Yaskawa INFORM job: vendrediTRJ1.JBI

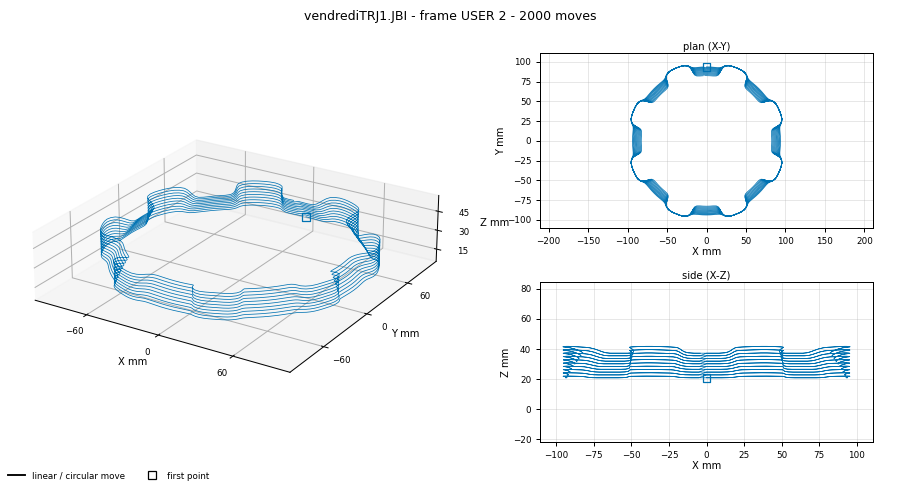
[picture p0: tool path of vendrediTRJ1.JBI in frame USER 2, 2000 of 2000 moves have a stored position in this frame; points joined in program order, loops and branches not executed]
/JOB
//NAME temp/vendrediTRJ1
///FOLDERNAME DEMO
//POS
///NPOS 2000,0,2000,0,0,0
///USER 2
///TOOL 7
///POSTYPE USER
///RECTAN
///RCONF 1,0,0,0,0,0,0,0,0,0,0,0,0,0,0,0,0,0,0,0,0,0,0,0
C00000=0.000,93.772,20.859,-180.0000,28.8281,-3690.0000
C00001=5.223,93.624,20.857,-179.9587,28.8401,-3693.1930
C00002=10.031,93.243,20.860,179.4696,28.7637,-3696.1402
C00003=14.399,92.874,20.935,176.5083,27.4530,-3698.8129
C00004=17.292,92.935,21.118,171.4736,22.1760,-3700.5402
C00005=19.271,93.399,21.361,170.6019,14.0567,-3701.6582
C00006=20.902,94.108,21.598,173.3176,8.0331,-3702.5225
C00007=22.556,94.852,21.773,176.3408,5.3244,-3703.3766
C00008=24.607,95.353,21.858,178.5800,3.6143,-3704.4702
C00009=27.423,95.407,21.902,179.6582,1.5415,-3706.0363
C00010=30.651,94.973,21.938,179.9852,0.1578,-3707.8866
C00011=33.828,94.073,21.973,-179.9998,0.0671,-3709.7782
C00012=36.813,92.974,21.997,179.9979,0.0053,-3711.6011
C00013=39.712,91.773,21.997,-179.9970,0.0075,-3713.3991
C00014=42.599,90.440,21.973,179.9991,0.0692,-3715.2213
C00015=45.483,88.829,21.938,-179.9836,0.1565,-3717.1138
C00016=48.072,86.854,21.902,-179.6591,1.5379,-3718.9637
C00017=50.025,84.825,21.858,-178.5802,3.6128,-3720.5297
C00018=51.121,83.020,21.773,-176.3413,5.3283,-3721.6234
C00019=51.765,81.324,21.598,-173.3148,8.0333,-3722.4779
C00020=52.416,79.670,21.361,-170.5989,14.0579,-3723.3415
C00021=53.488,77.942,21.118,-171.4764,22.1779,-3724.4600
C00022=55.491,75.854,20.935,-176.5044,27.4539,-3726.1873
C00023=58.840,73.026,20.860,-179.4708,28.7627,-3728.8598
C00024=62.509,69.895,20.857,179.9582,28.8407,-3731.8071
C00025=66.307,66.307,20.859,180.0000,28.8305,-3735.0000
C00026=69.895,62.509,20.857,-179.9582,28.8407,-3738.1929
C00027=73.026,58.840,20.860,179.4708,28.7627,-3741.1402
C00028=75.854,55.491,20.935,176.5044,27.4539,-3743.8127
C00029=77.942,53.488,21.118,171.4764,22.1779,-3745.5400
C00030=79.670,52.416,21.361,170.5989,14.0579,-3746.6585
C00031=81.324,51.765,21.598,173.3148,8.0333,-3747.5221
C00032=83.020,51.121,21.773,176.3413,5.3283,-3748.3766
C00033=84.825,50.025,21.858,178.5802,3.6128,-3749.4703
C00034=86.854,48.072,21.902,179.6591,1.5379,-3751.0363
C00035=88.829,45.483,21.938,179.9836,0.1565,-3752.8862
C00036=90.440,42.599,21.973,-179.9991,0.0692,-3754.7787
C00037=91.773,39.712,21.997,179.9970,0.0075,-3756.6009
C00038=92.974,36.813,21.997,-179.9979,0.0053,-3758.3989
C00039=94.073,33.828,21.973,179.9998,0.0671,-3760.2218
C00040=94.973,30.651,21.938,-179.9852,0.1578,-3762.1134
C00041=95.407,27.423,21.902,-179.6582,1.5415,-3763.9637
C00042=95.353,24.607,21.858,-178.5800,3.6143,-3765.5298
C00043=94.852,22.556,21.773,-176.3408,5.3244,-3766.6234
C00044=94.108,20.902,21.598,-173.3176,8.0331,-3767.4775
C00045=93.399,19.271,21.361,-170.6019,14.0567,-3768.3418
C00046=92.935,17.292,21.118,-171.4736,22.1760,-3769.4598
C00047=92.874,14.399,20.935,-176.5083,27.4530,-3771.1871
C00048=93.243,10.031,20.860,-179.4696,28.7637,-3773.8598
C00049=93.624,5.223,20.857,179.9587,28.8401,-3776.8070
C00050=93.772,0.000,20.859,180.0000,28.8281,-3780.0000
C00051=93.624,-5.223,20.857,-179.9587,28.8401,-3783.1930
C00052=93.243,-10.031,20.860,179.4696,28.7637,-3786.1402
C00053=92.875,-14.399,20.935,176.5083,27.4530,-3788.8128
C00054=92.935,-17.292,21.118,171.4736,22.1760,-3790.5402
C00055=93.399,-19.271,21.361,170.6019,14.0567,-3791.6582
C00056=94.108,-20.902,21.598,173.3176,8.0331,-3792.5225
C00057=94.852,-22.556,21.773,176.3408,5.3244,-3793.3766
C00058=95.353,-24.607,21.858,178.5800,3.6143,-3794.4702
C00059=95.407,-27.423,21.902,179.6582,1.5415,-3796.0363
C00060=94.973,-30.651,21.938,179.9852,0.1578,-3797.8866
C00061=94.073,-33.828,21.973,-179.9998,0.0671,-3799.7782
C00062=92.974,-36.813,21.997,179.9979,0.0053,-3801.6011
C00063=91.773,-39.712,21.997,-179.9970,0.0075,-3803.3991
C00064=90.440,-42.599,21.973,179.9991,0.0692,-3805.2213
C00065=88.829,-45.483,21.938,-179.9836,0.1565,-3807.1138
C00066=86.854,-48.072,21.902,-179.6591,1.5379,-3808.9637
C00067=84.825,-50.025,21.858,-178.5802,3.6128,-3810.5297
C00068=83.020,-51.121,21.773,-176.3413,5.3283,-3811.6234
C00069=81.324,-51.765,21.598,-173.3148,8.0333,-3812.4779
C00070=79.670,-52.416,21.361,-170.5989,14.0579,-3813.3415
C00071=77.942,-53.488,21.118,-171.4764,22.1779,-3814.4600
C00072=75.854,-55.491,20.935,-176.5044,27.4539,-3816.1873
C00073=73.026,-58.840,20.860,-179.4708,28.7627,-3818.8598
C00074=69.895,-62.509,20.857,179.9582,28.8407,-3821.8071
C00075=66.307,-66.307,20.859,-180.0000,28.8305,-3825.0000
C00076=62.509,-69.895,20.857,-179.9582,28.8407,-3828.1929
C00077=58.840,-73.026,20.860,179.4708,28.7627,-3831.1402
C00078=55.491,-75.854,20.935,176.5044,27.4539,-3833.8127
C00079=53.488,-77.942,21.118,171.4764,22.1779,-3835.5400
C00080=52.416,-79.670,21.361,170.5989,14.0579,-3836.6585
C00081=51.765,-81.324,21.598,173.3148,8.0333,-3837.5221
C00082=51.121,-83.020,21.773,176.3413,5.3283,-3838.3766
C00083=50.025,-84.825,21.858,178.5802,3.6128,-3839.4703
C00084=48.072,-86.854,21.902,179.6591,1.5379,-3841.0363
C00085=45.483,-88.829,21.938,179.9836,0.1565,-3842.8862
C00086=42.599,-90.440,21.973,-179.9991,0.0692,-3844.7787
C00087=39.712,-91.773,21.997,179.9970,0.0075,-3846.6009
C00088=36.813,-92.974,21.997,-179.9979,0.0053,-3848.3989
C00089=33.828,-94.073,21.973,179.9998,0.0671,-3850.2218
C00090=30.651,-94.973,21.938,-179.9852,0.1578,-3852.1134
C00091=27.423,-95.407,21.902,-179.6582,1.5415,-3853.9637
C00092=24.607,-95.353,21.858,-178.5800,3.6143,-3855.5298
C00093=22.556,-94.852,21.773,-176.3408,5.3244,-3856.6234
C00094=20.902,-94.108,21.598,-173.3176,8.0331,-3857.4775
C00095=19.271,-93.399,21.361,-170.6019,14.0567,-3858.3418
C00096=17.292,-92.935,21.118,-171.4736,22.1760,-3859.4598
C00097=14.399,-92.874,20.935,-176.5083,27.4530,-3861.1871
C00098=10.031,-93.243,20.860,-179.4696,28.7637,-3863.8598
C00099=5.223,-93.624,20.857,179.9587,28.8401,-3866.8070
C00100=0.000,-93.772,20.859,-180.0000,28.8281,-3870.0000
C00101=-5.223,-93.624,20.857,-179.9587,28.8401,-3873.1930
C00102=-10.031,-93.243,20.860,179.4696,28.7637,-3876.1402
C00103=-14.399,-92.875,20.935,176.5083,27.4530,-3878.8128
C00104=-17.292,-92.935,21.118,171.4736,22.1760,-3880.5402
C00105=-19.271,-93.399,21.361,170.6019,14.0567,-3881.6582
C00106=-20.902,-94.108,21.598,173.3176,8.0331,-3882.5225
C00107=-22.556,-94.852,21.773,176.3408,5.3244,-3883.3766
C00108=-24.607,-95.353,21.858,178.5800,3.6143,-3884.4702
C00109=-27.423,-95.407,21.902,179.6582,1.5415,-3886.0363
C00110=-30.651,-94.973,21.938,179.9852,0.1578,-3887.8866
C00111=-33.828,-94.073,21.973,-179.9998,0.0671,-3889.7782
C00112=-36.813,-92.974,21.997,179.9979,0.0053,-3891.6011
C00113=-39.712,-91.773,21.997,-179.9970,0.0075,-3893.3991
C00114=-42.599,-90.440,21.973,179.9991,0.0692,-3895.2213
C00115=-45.483,-88.829,21.938,-179.9836,0.1565,-3897.1138
C00116=-48.072,-86.854,21.902,-179.6591,1.5379,-3898.9637
C00117=-50.025,-84.825,21.858,-178.5802,3.6128,-3900.5297
C00118=-51.121,-83.020,21.773,-176.3413,5.3283,-3901.6234
C00119=-51.765,-81.324,21.598,-173.3148,8.0333,-3902.4779
C00120=-52.416,-79.670,21.361,-170.5989,14.0579,-3903.3415
C00121=-53.488,-77.942,21.118,-171.4764,22.1779,-3904.4600
C00122=-55.491,-75.854,20.935,-176.5044,27.4539,-3906.1873
C00123=-58.840,-73.026,20.860,-179.4708,28.7627,-3908.8598
C00124=-62.509,-69.895,20.857,179.9582,28.8407,-3911.8071
C00125=-66.307,-66.307,20.859,-180.0000,28.8305,-3915.0000
C00126=-69.895,-62.509,20.857,-179.9582,28.8407,-3918.1929
C00127=-73.026,-58.840,20.860,179.4708,28.7627,-3921.1402
C00128=-75.854,-55.491,20.935,176.5044,27.4539,-3923.8127
C00129=-77.942,-53.488,21.118,171.4764,22.1779,-3925.5400
C00130=-79.670,-52.416,21.361,170.5989,14.0579,-3926.6585
C00131=-81.324,-51.765,21.598,173.3148,8.0333,-3927.5221
C00132=-83.020,-51.121,21.773,176.3413,5.3283,-3928.3766
C00133=-84.825,-50.025,21.858,178.5802,3.6128,-3929.4703
C00134=-86.854,-48.072,21.902,179.6591,1.5379,-3931.0363
C00135=-88.829,-45.483,21.938,179.9836,0.1565,-3932.8862
C00136=-90.440,-42.599,21.973,-179.9991,0.0692,-3934.7787
C00137=-91.773,-39.712,21.997,179.9970,0.0075,-3936.6009
C00138=-92.974,-36.813,21.997,-179.9979,0.0053,-3938.3989
C00139=-94.073,-33.828,21.973,179.9998,0.0671,-3940.2218
C00140=-94.973,-30.651,21.938,-179.9852,0.1578,-3942.1134
C00141=-95.407,-27.423,21.902,-179.6582,1.5415,-3943.9637
C00142=-95.353,-24.607,21.858,-178.5800,3.6143,-3945.5298
C00143=-94.852,-22.556,21.773,-176.3408,5.3244,-3946.6234
C00144=-94.108,-20.902,21.598,-173.3176,8.0331,-3947.4775
C00145=-93.399,-19.271,21.361,-170.6019,14.0567,-3948.3418
C00146=-92.935,-17.292,21.118,-171.4736,22.1760,-3949.4598
C00147=-92.874,-14.399,20.935,-176.5083,27.4530,-3951.1871
C00148=-93.243,-10.031,20.860,-179.4696,28.7637,-3953.8598
C00149=-93.624,-5.223,20.857,179.9587,28.8401,-3956.8070
C00150=-93.772,0.000,20.859,180.0000,28.8281,-3960.0000
C00151=-93.624,5.223,20.857,-179.9587,28.8401,-3963.1930
C00152=-93.243,10.031,20.860,179.4696,28.7637,-3966.1402
C00153=-92.875,14.399,20.935,176.5083,27.4530,-3968.8128
C00154=-92.935,17.292,21.118,171.4736,22.1760,-3970.5402
C00155=-93.399,19.271,21.361,170.6019,14.0567,-3971.6582
C00156=-94.108,20.902,21.598,173.3176,8.0331,-3972.5225
C00157=-94.852,22.556,21.773,176.3408,5.3244,-3973.3766
C00158=-95.353,24.607,21.858,178.5800,3.6143,-3974.4702
C00159=-95.407,27.423,21.902,179.6582,1.5415,-3976.0363
C00160=-94.973,30.651,21.938,179.9852,0.1578,-3977.8866
C00161=-94.073,33.828,21.973,-179.9998,0.0671,-3979.7782
C00162=-92.974,36.813,21.997,179.9979,0.0053,-3981.6011
C00163=-91.773,39.712,21.997,-179.9970,0.0075,-3983.3991
C00164=-90.440,42.599,21.973,179.9991,0.0692,-3985.2213
C00165=-88.829,45.483,21.938,-179.9836,0.1565,-3987.1138
C00166=-86.854,48.072,21.902,-179.6591,1.5379,-3988.9637
C00167=-84.825,50.025,21.858,-178.5802,3.6128,-3990.5297
C00168=-83.020,51.121,21.773,-176.3413,5.3283,-3991.6234
C00169=-81.324,51.765,21.598,-173.3148,8.0333,-3992.4779
C00170=-79.670,52.416,21.361,-170.5989,14.0579,-3993.3415
C00171=-77.942,53.488,21.118,-171.4764,22.1779,-3994.4600
C00172=-75.854,55.491,20.935,-176.5044,27.4539,-3996.1873
C00173=-73.026,58.840,20.860,-179.4708,28.7627,-3998.8598
C00174=-69.895,62.509,20.857,179.9582,28.8407,-4001.8071
C00175=-66.307,66.307,20.859,180.0000,28.8305,-4005.0000
C00176=-62.509,69.895,20.857,-179.9582,28.8407,-4008.1929
C00177=-58.840,73.026,20.860,179.4708,28.7627,-4011.1402
C00178=-55.491,75.854,20.935,176.5044,27.4539,-4013.8127
C00179=-53.488,77.942,21.118,171.4764,22.1779,-4015.5400
C00180=-52.416,79.670,21.361,170.5989,14.0579,-4016.6585
C00181=-51.765,81.324,21.598,173.3148,8.0333,-4017.5221
C00182=-51.121,83.020,21.773,176.3413,5.3283,-4018.3766
C00183=-50.025,84.825,21.858,178.5802,3.6128,-4019.4703
C00184=-48.072,86.854,21.902,179.6591,1.5379,-4021.0363
C00185=-45.483,88.829,21.938,179.9836,0.1565,-4022.8862
C00186=-42.599,90.440,21.973,-179.9991,0.0692,-4024.7787
C00187=-39.712,91.773,21.997,179.9970,0.0075,-4026.6009
C00188=-36.813,92.974,21.997,-179.9979,0.0053,-4028.3989
C00189=-33.828,94.073,21.973,179.9998,0.0671,-4030.2218
C00190=-30.651,94.973,21.938,-179.9852,0.1578,-4032.1134
C00191=-27.423,95.407,21.902,-179.6582,1.5415,-4033.9637
C00192=-24.607,95.353,21.858,-178.5800,3.6143,-4035.5298
C00193=-22.556,94.852,21.773,-176.3408,5.3244,-4036.6234
C00194=-20.902,94.108,21.598,-173.3176,8.0331,-4037.4775
C00195=-19.271,93.399,21.361,-170.6019,14.0567,-4038.3418
C00196=-17.292,92.935,21.118,-171.4736,22.1760,-4039.4598
C00197=-14.399,92.875,20.935,-176.5083,27.4530,-4041.1872
C00198=-10.031,93.243,20.860,-179.4696,28.7637,-4043.8598
C00199=-5.223,93.624,20.857,179.9587,28.8401,-4046.8070
C00200=0.000,92.684,22.771,-180.0000,30.3909,-4050.0000
C00201=5.124,92.540,22.769,-179.9518,30.3994,-4053.1693
C00202=9.864,92.169,22.773,179.3255,30.3134,-4056.1086
C00203=14.194,91.838,22.865,175.6033,28.8062,-4058.7858
C00204=17.042,91.994,23.091,169.6619,22.2216,-4060.4951
C00205=18.986,92.606,23.393,169.6266,12.7358,-4061.5862
C00206=20.592,93.503,23.691,173.2393,6.5920,-4062.4199
C00207=22.223,94.456,23.912,176.4053,4.2313,-4063.2394
C00208=24.245,95.156,24.019,178.5515,3.0336,-4064.2944
C00209=27.082,95.366,24.075,179.6706,1.2647,-4065.8535
C00210=30.380,95.022,24.120,179.9985,0.0236,-4067.7299
C00211=33.658,94.129,24.166,179.9969,0.0597,-4069.6757
C00212=36.755,92.996,24.196,179.9979,0.0053,-4071.5655
C00213=39.769,91.748,24.196,179.9977,0.0053,-4073.4348
C00214=42.760,90.359,24.166,179.9987,0.0564,-4075.3246
C00215=45.709,88.673,24.120,-179.9977,0.0205,-4077.2701
C00216=48.284,86.584,24.075,-179.6697,1.2668,-4079.1464
C00217=50.142,84.429,24.019,-178.5525,3.0331,-4080.7059
C00218=51.076,82.504,23.912,-176.4065,4.2307,-4081.7605
C00219=51.556,80.678,23.691,-173.2418,6.5908,-4082.5800
C00220=52.057,78.907,23.393,-169.6292,12.7370,-4083.4139
C00221=52.999,77.101,23.091,-169.6605,22.2236,-4084.5045
C00222=54.903,74.976,22.865,-175.5993,28.8036,-4086.2144
C00223=58.198,72.148,22.773,-179.3268,30.3167,-4088.8913
C00224=61.813,69.059,22.769,179.9465,30.4010,-4091.8309
C00225=65.538,65.538,22.771,-180.0000,30.3891,-4095.0000
C00226=69.059,61.813,22.769,-179.9465,30.4010,-4098.1691
C00227=72.148,58.198,22.773,179.3268,30.3167,-4101.1087
C00228=74.976,54.903,22.865,175.6032,28.8076,-4103.7856
C00229=77.101,52.999,23.091,169.6605,22.2236,-4105.4955
C00230=78.907,52.057,23.393,169.6292,12.7370,-4106.5861
C00231=80.678,51.556,23.691,173.2418,6.5908,-4107.4200
C00232=82.504,51.076,23.912,176.4065,4.2307,-4108.2395
C00233=84.429,50.142,24.019,178.5525,3.0331,-4109.2941
C00234=86.584,48.284,24.075,179.6697,1.2668,-4110.8536
C00235=88.673,45.709,24.120,179.9977,0.0205,-4112.7299
C00236=90.359,42.760,24.166,-179.9987,0.0564,-4114.6754
C00237=91.748,39.769,24.196,-179.9977,0.0053,-4116.5652
C00238=92.996,36.755,24.196,-179.9979,0.0053,-4118.4345
C00239=94.129,33.658,24.166,-179.9969,0.0597,-4120.3243
C00240=95.022,30.380,24.120,-179.9985,0.0236,-4122.2701
C00241=95.366,27.082,24.075,-179.6706,1.2647,-4124.1465
C00242=95.156,24.245,24.019,-178.5515,3.0336,-4125.7056
C00243=94.456,22.223,23.912,-176.4053,4.2313,-4126.7606
C00244=93.503,20.592,23.691,-173.2393,6.5920,-4127.5801
C00245=92.606,18.986,23.393,-169.6266,12.7358,-4128.4138
C00246=91.994,17.042,23.091,-169.6619,22.2216,-4129.5049
C00247=91.838,14.194,22.865,-175.6033,28.8062,-4131.2142
C00248=92.169,9.864,22.773,-179.3255,30.3134,-4133.8914
C00249=92.540,5.124,22.769,179.9518,30.3994,-4136.8307
C00250=92.684,0.000,22.771,-180.0000,30.3909,-4140.0000
C00251=92.540,-5.124,22.769,-179.9518,30.3994,-4143.1693
C00252=92.169,-9.864,22.773,179.3255,30.3134,-4146.1086
C00253=91.838,-14.194,22.865,175.6033,28.8062,-4148.7858
C00254=91.994,-17.042,23.091,169.6619,22.2216,-4150.4951
C00255=92.606,-18.986,23.393,169.6266,12.7358,-4151.5862
C00256=93.503,-20.592,23.691,173.2393,6.5920,-4152.4199
C00257=94.456,-22.223,23.912,176.4053,4.2313,-4153.2394
C00258=95.156,-24.245,24.019,178.5515,3.0336,-4154.2944
C00259=95.366,-27.082,24.075,179.6706,1.2647,-4155.8535
C00260=95.022,-30.380,24.120,179.9985,0.0236,-4157.7299
C00261=94.129,-33.658,24.166,179.9969,0.0597,-4159.6757
C00262=92.996,-36.755,24.196,179.9979,0.0053,-4161.5655
C00263=91.748,-39.769,24.196,179.9977,0.0053,-4163.4348
C00264=90.359,-42.760,24.166,179.9987,0.0564,-4165.3246
C00265=88.673,-45.709,24.120,-179.9977,0.0205,-4167.2701
C00266=86.584,-48.284,24.075,-179.6697,1.2668,-4169.1464
C00267=84.429,-50.142,24.019,-178.5525,3.0331,-4170.7059
C00268=82.504,-51.076,23.912,-176.4065,4.2307,-4171.7605
C00269=80.678,-51.556,23.691,-173.2418,6.5908,-4172.5800
C00270=78.907,-52.057,23.393,-169.6292,12.7370,-4173.4139
C00271=77.101,-52.999,23.091,-169.6605,22.2236,-4174.5045
C00272=74.976,-54.903,22.865,-175.5993,28.8036,-4176.2144
C00273=72.148,-58.198,22.773,-179.3268,30.3167,-4178.8913
C00274=69.059,-61.813,22.769,179.9465,30.4010,-4181.8309
C00275=65.538,-65.538,22.771,180.0000,30.3891,-4185.0000
C00276=61.813,-69.059,22.769,-179.9465,30.4010,-4188.1691
C00277=58.198,-72.148,22.773,179.3268,30.3167,-4191.1087
C00278=54.903,-74.976,22.865,175.6032,28.8076,-4193.7856
C00279=52.999,-77.101,23.091,169.6605,22.2236,-4195.4955
C00280=52.057,-78.907,23.393,169.6292,12.7370,-4196.5861
C00281=51.556,-80.678,23.691,173.2418,6.5908,-4197.4200
C00282=51.076,-82.504,23.912,176.4065,4.2307,-4198.2395
C00283=50.142,-84.429,24.019,178.5525,3.0331,-4199.2941
C00284=48.284,-86.584,24.075,179.6697,1.2668,-4200.8536
C00285=45.709,-88.673,24.120,179.9977,0.0205,-4202.7299
C00286=42.760,-90.359,24.166,-179.9987,0.0564,-4204.6754
C00287=39.769,-91.748,24.196,-179.9977,0.0053,-4206.5652
C00288=36.755,-92.996,24.196,-179.9979,0.0053,-4208.4345
C00289=33.658,-94.129,24.166,-179.9969,0.0597,-4210.3243
C00290=30.380,-95.022,24.120,-179.9985,0.0236,-4212.2701
C00291=27.082,-95.366,24.075,-179.6706,1.2647,-4214.1465
C00292=24.245,-95.156,24.019,-178.5515,3.0336,-4215.7056
C00293=22.223,-94.456,23.912,-176.4053,4.2313,-4216.7606
C00294=20.592,-93.503,23.691,-173.2393,6.5920,-4217.5801
C00295=18.986,-92.606,23.393,-169.6266,12.7358,-4218.4138
C00296=17.042,-91.994,23.091,-169.6619,22.2216,-4219.5049
C00297=14.194,-91.838,22.865,-175.6033,28.8062,-4221.2142
C00298=9.864,-92.169,22.773,-179.3255,30.3134,-4223.8914
C00299=5.124,-92.540,22.769,179.9518,30.3994,-4226.8307
C00300=0.000,-92.684,22.771,180.0000,30.3909,-4230.0000
C00301=-5.124,-92.540,22.769,-179.9518,30.3994,-4233.1693
C00302=-9.864,-92.169,22.773,179.3255,30.3134,-4236.1086
C00303=-14.194,-91.838,22.865,175.6033,28.8062,-4238.7858
C00304=-17.042,-91.994,23.091,169.6619,22.2216,-4240.4951
C00305=-18.986,-92.606,23.393,169.6266,12.7358,-4241.5862
C00306=-20.592,-93.503,23.691,173.2393,6.5920,-4242.4199
C00307=-22.223,-94.456,23.912,176.4053,4.2313,-4243.2394
C00308=-24.245,-95.156,24.019,178.5515,3.0336,-4244.2944
C00309=-27.082,-95.366,24.075,179.6706,1.2647,-4245.8535
C00310=-30.380,-95.022,24.120,179.9985,0.0236,-4247.7299
C00311=-33.658,-94.129,24.166,179.9969,0.0597,-4249.6757
C00312=-36.755,-92.996,24.196,179.9979,0.0053,-4251.5655
C00313=-39.769,-91.748,24.196,179.9977,0.0053,-4253.4348
C00314=-42.760,-90.359,24.166,179.9987,0.0564,-4255.3246
C00315=-45.709,-88.673,24.120,-179.9977,0.0205,-4257.2701
C00316=-48.284,-86.584,24.075,-179.6697,1.2668,-4259.1464
C00317=-50.142,-84.429,24.019,-178.5525,3.0331,-4260.7059
C00318=-51.076,-82.504,23.912,-176.4065,4.2307,-4261.7605
C00319=-51.556,-80.678,23.691,-173.2418,6.5908,-4262.5800
C00320=-52.057,-78.907,23.393,-169.6292,12.7370,-4263.4139
C00321=-52.999,-77.101,23.091,-169.6605,22.2236,-4264.5045
C00322=-54.903,-74.976,22.865,-175.5993,28.8036,-4266.2144
C00323=-58.198,-72.148,22.773,-179.3268,30.3167,-4268.8913
C00324=-61.813,-69.059,22.769,179.9465,30.4010,-4271.8309
C00325=-65.538,-65.538,22.771,-180.0000,30.3891,-4275.0000
C00326=-69.059,-61.813,22.769,-179.9465,30.4010,-4278.1691
C00327=-72.148,-58.198,22.773,179.3268,30.3167,-4281.1087
C00328=-74.976,-54.903,22.865,175.6032,28.8076,-4283.7856
C00329=-77.101,-52.999,23.091,169.6605,22.2236,-4285.4955
C00330=-78.907,-52.057,23.393,169.6292,12.7370,-4286.5861
C00331=-80.678,-51.556,23.691,173.2418,6.5908,-4287.4200
C00332=-82.504,-51.076,23.912,176.4065,4.2307,-4288.2395
C00333=-84.429,-50.142,24.019,178.5525,3.0331,-4289.2941
C00334=-86.584,-48.284,24.075,179.6697,1.2668,-4290.8536
C00335=-88.673,-45.709,24.120,179.9977,0.0205,-4292.7299
C00336=-90.359,-42.760,24.166,-179.9987,0.0564,-4294.6754
C00337=-91.748,-39.769,24.196,-179.9977,0.0053,-4296.5652
C00338=-92.996,-36.755,24.196,-179.9979,0.0053,-4298.4345
C00339=-94.129,-33.658,24.166,-179.9969,0.0597,-4300.3243
C00340=-95.022,-30.380,24.120,-179.9985,0.0236,-4302.2701
C00341=-95.366,-27.082,24.075,-179.6706,1.2647,-4304.1465
C00342=-95.156,-24.245,24.019,-178.5515,3.0336,-4305.7056
C00343=-94.456,-22.223,23.912,-176.4053,4.2313,-4306.7606
C00344=-93.503,-20.592,23.691,-173.2393,6.5920,-4307.5801
C00345=-92.606,-18.986,23.393,-169.6266,12.7358,-4308.4138
C00346=-91.994,-17.042,23.091,-169.6619,22.2216,-4309.5049
C00347=-91.838,-14.194,22.865,-175.6033,28.8062,-4311.2142
C00348=-92.169,-9.864,22.773,-179.3255,30.3134,-4313.8914
C00349=-92.540,-5.124,22.769,179.9518,30.3994,-4316.8307
C00350=-92.684,0.000,22.771,-180.0000,30.3909,-4320.0000
C00351=-92.540,5.124,22.769,-179.9518,30.3994,-4323.1693
C00352=-92.169,9.864,22.773,179.3255,30.3134,-4326.1086
C00353=-91.838,14.194,22.865,175.6033,28.8062,-4328.7858
C00354=-91.994,17.042,23.091,169.6619,22.2216,-4330.4951
C00355=-92.606,18.986,23.393,169.6266,12.7358,-4331.5862
C00356=-93.503,20.592,23.691,173.2393,6.5920,-4332.4199
C00357=-94.456,22.223,23.912,176.4053,4.2313,-4333.2394
C00358=-95.156,24.245,24.019,178.5515,3.0336,-4334.2944
C00359=-95.366,27.082,24.075,179.6706,1.2647,-4335.8535
C00360=-95.022,30.380,24.120,179.9985,0.0236,-4337.7299
C00361=-94.129,33.658,24.166,179.9969,0.0597,-4339.6757
C00362=-92.996,36.755,24.196,179.9979,0.0053,-4341.5655
C00363=-91.748,39.769,24.196,179.9977,0.0053,-4343.4348
C00364=-90.359,42.760,24.166,179.9987,0.0564,-4345.3246
C00365=-88.673,45.709,24.120,-179.9977,0.0205,-4347.2701
C00366=-86.584,48.284,24.075,-179.6697,1.2668,-4349.1464
C00367=-84.429,50.142,24.019,-178.5525,3.0331,-4350.7059
C00368=-82.504,51.076,23.912,-176.4065,4.2307,-4351.7605
C00369=-80.678,51.556,23.691,-173.2418,6.5908,-4352.5800
C00370=-78.907,52.057,23.393,-169.6292,12.7370,-4353.4139
C00371=-77.101,52.999,23.091,-169.6605,22.2236,-4354.5045
C00372=-74.976,54.903,22.865,-175.5993,28.8036,-4356.2144
C00373=-72.148,58.198,22.773,-179.3268,30.3167,-4358.8913
C00374=-69.059,61.813,22.769,179.9465,30.4010,-4361.8309
C00375=-65.538,65.538,22.771,-180.0000,30.3891,-4365.0000
C00376=-61.813,69.059,22.769,-179.9465,30.4010,-4368.1691
C00377=-58.198,72.148,22.773,179.3268,30.3167,-4371.1087
C00378=-54.903,74.976,22.865,175.6032,28.8076,-4373.7856
C00379=-52.999,77.101,23.091,169.6605,22.2236,-4375.4955
C00380=-52.057,78.907,23.393,169.6292,12.7370,-4376.5861
C00381=-51.556,80.678,23.691,173.2418,6.5908,-4377.4200
C00382=-51.076,82.504,23.912,176.4065,4.2307,-4378.2395
C00383=-50.142,84.429,24.019,178.5525,3.0331,-4379.2941
C00384=-48.284,86.584,24.075,179.6697,1.2668,-4380.8536
C00385=-45.709,88.673,24.120,179.9977,0.0205,-4382.7299
C00386=-42.760,90.359,24.166,-179.9987,0.0564,-4384.6754
C00387=-39.769,91.748,24.196,-179.9977,0.0053,-4386.5652
C00388=-36.755,92.996,24.196,-179.9979,0.0053,-4388.4345
C00389=-33.658,94.129,24.166,-179.9969,0.0597,-4390.3243
C00390=-30.380,95.022,24.120,-179.9985,0.0236,-4392.2701
C00391=-27.082,95.366,24.075,-179.6706,1.2647,-4394.1465
C00392=-24.245,95.156,24.019,-178.5515,3.0336,-4395.7056
C00393=-22.223,94.456,23.912,-176.4053,4.2313,-4396.7606
C00394=-20.592,93.503,23.691,-173.2393,6.5920,-4397.5801
C00395=-18.986,92.606,23.393,-169.6266,12.7358,-4398.4138
C00396=-17.042,91.994,23.091,-169.6619,22.2216,-4399.5049
C00397=-14.194,91.838,22.865,-175.6033,28.8062,-4401.2142
C00398=-9.864,92.169,22.773,-179.3255,30.3134,-4403.8914
C00399=-5.124,92.540,22.769,179.9518,30.3994,-4406.8307
C00400=0.000,91.548,24.655,-180.0000,31.7764,-4410.0000
C00401=5.020,91.408,24.652,-179.9386,31.7913,-4413.1434
C00402=9.690,91.047,24.657,179.1672,31.6940,-4416.0750
C00403=13.981,90.755,24.767,174.6081,29.9498,-4418.7577
C00404=16.781,91.008,25.041,167.9432,21.7872,-4420.4474
C00405=18.686,91.772,25.406,169.1360,11.0995,-4421.5089
C00406=20.265,92.865,25.771,173.6100,5.1205,-4422.3101
C00407=21.871,94.037,26.043,176.8157,3.0731,-4423.0930
C00408=23.861,94.948,26.175,178.6786,2.3162,-4424.1066
C00409=26.720,95.323,26.245,179.7166,0.9262,-4425.6587
C00410=30.093,95.074,26.301,-179.9821,-0.1326,-4427.5637
C00411=33.476,94.189,26.358,-179.9972,0.0435,-4429.5659
C00412=36.693,93.020,26.395,179.9979,0.0053,-4431.5274
C00413=39.829,91.721,26.395,179.9977,0.0053,-4433.4725
C00414=42.931,90.273,26.358,179.9983,0.0436,-4435.4343
C00415=45.948,88.507,26.301,179.9790,-0.1336,-4437.4359
C00416=48.509,86.297,26.245,-179.7191,0.9269,-4439.3411
C00417=50.266,84.010,26.175,-178.6733,2.3167,-4440.8935
C00418=51.029,81.959,26.043,-176.8139,3.0727,-4441.9071
C00419=51.336,79.995,25.771,-173.6111,5.1213,-4442.6899
C00420=51.679,78.105,25.406,-169.1359,11.0962,-4443.4910
C00421=52.487,76.218,25.041,-167.9434,21.7869,-4444.5530
C00422=54.287,74.059,24.767,-174.6079,29.9481,-4446.2423
C00423=57.528,71.231,24.657,-179.1658,31.6931,-4448.9252
C00424=61.085,68.184,24.652,179.9356,31.7887,-4451.8567
C00425=64.734,64.734,24.655,180.0000,31.7790,-4455.0000
C00426=68.184,61.085,24.652,-179.9356,31.7887,-4458.1433
C00427=71.231,57.528,24.657,179.1658,31.6931,-4461.0748
C00428=74.059,54.287,24.767,174.6079,29.9481,-4463.7577
C00429=76.218,52.487,25.041,167.9434,21.7869,-4465.4470
C00430=78.105,51.679,25.406,169.1359,11.0962,-4466.5090
C00431=79.995,51.336,25.771,173.6111,5.1213,-4467.3101
C00432=81.959,51.029,26.043,176.8139,3.0727,-4468.0929
C00433=84.010,50.266,26.175,178.6733,2.3167,-4469.1065
C00434=86.297,48.509,26.245,179.7191,0.9269,-4470.6589
C00435=88.507,45.948,26.301,-179.9790,-0.1336,-4472.5641
C00436=90.273,42.931,26.358,-179.9983,0.0436,-4474.5657
C00437=91.721,39.829,26.395,-179.9977,0.0053,-4476.5275
C00438=93.020,36.693,26.395,-179.9979,0.0053,-4478.4726
C00439=94.189,33.476,26.358,179.9972,0.0435,-4480.4341
C00440=95.074,30.093,26.301,179.9821,-0.1326,-4482.4363
C00441=95.323,26.720,26.245,-179.7166,0.9262,-4484.3413
C00442=94.948,23.861,26.175,-178.6786,2.3162,-4485.8934
C00443=94.037,21.871,26.043,-176.8157,3.0731,-4486.9070
C00444=92.865,20.265,25.771,-173.6100,5.1205,-4487.6899
C00445=91.772,18.686,25.406,-169.1360,11.0995,-4488.4911
C00446=91.008,16.781,25.041,-167.9432,21.7872,-4489.5526
C00447=90.755,13.981,24.767,-174.6081,29.9498,-4491.2423
C00448=91.047,9.690,24.657,-179.1672,31.6940,-4493.9250
C00449=91.408,5.020,24.652,179.9386,31.7913,-4496.8566
C00450=91.548,0.000,24.655,180.0000,31.7764,-4500.0000
C00451=91.408,-5.020,24.652,-179.9386,31.7913,-4503.1434
C00452=91.047,-9.690,24.657,179.1672,31.6940,-4506.0750
C00453=90.755,-13.981,24.767,174.6081,29.9498,-4508.7577
C00454=91.008,-16.781,25.041,167.9432,21.7872,-4510.4474
C00455=91.772,-18.686,25.406,169.1360,11.0995,-4511.5089
C00456=92.865,-20.265,25.771,173.6100,5.1205,-4512.3101
C00457=94.037,-21.871,26.043,176.8157,3.0731,-4513.0930
C00458=94.948,-23.861,26.175,178.6786,2.3162,-4514.1066
C00459=95.323,-26.720,26.245,179.7166,0.9262,-4515.6587
C00460=95.074,-30.093,26.301,-179.9821,-0.1326,-4517.5637
C00461=94.189,-33.476,26.358,-179.9972,0.0435,-4519.5659
C00462=93.020,-36.693,26.395,179.9979,0.0053,-4521.5274
C00463=91.721,-39.829,26.395,179.9977,0.0053,-4523.4725
C00464=90.273,-42.931,26.358,179.9983,0.0436,-4525.4343
C00465=88.507,-45.948,26.301,179.9790,-0.1336,-4527.4359
C00466=86.297,-48.509,26.245,-179.7191,0.9269,-4529.3411
C00467=84.010,-50.266,26.175,-178.6733,2.3167,-4530.8935
C00468=81.959,-51.029,26.043,-176.8139,3.0727,-4531.9071
C00469=79.995,-51.336,25.771,-173.6111,5.1213,-4532.6899
C00470=78.105,-51.679,25.406,-169.1359,11.0962,-4533.4910
C00471=76.218,-52.487,25.041,-167.9434,21.7869,-4534.5530
C00472=74.059,-54.287,24.767,-174.6079,29.9481,-4536.2423
C00473=71.231,-57.528,24.657,-179.1658,31.6931,-4538.9252
C00474=68.184,-61.085,24.652,179.9356,31.7887,-4541.8567
C00475=64.734,-64.734,24.655,-180.0000,31.7790,-4545.0000
C00476=61.085,-68.184,24.652,-179.9356,31.7887,-4548.1433
C00477=57.528,-71.231,24.657,179.1658,31.6931,-4551.0748
C00478=54.287,-74.059,24.767,174.6079,29.9481,-4553.7577
C00479=52.487,-76.218,25.041,167.9434,21.7869,-4555.4470
C00480=51.679,-78.105,25.406,169.1359,11.0962,-4556.5090
C00481=51.336,-79.995,25.771,173.6111,5.1213,-4557.3101
C00482=51.029,-81.959,26.043,176.8139,3.0727,-4558.0929
C00483=50.266,-84.010,26.175,178.6733,2.3167,-4559.1065
C00484=48.509,-86.297,26.245,179.7191,0.9269,-4560.6589
C00485=45.948,-88.507,26.301,-179.9790,-0.1336,-4562.5641
C00486=42.931,-90.273,26.358,-179.9983,0.0436,-4564.5657
C00487=39.829,-91.721,26.395,-179.9977,0.0053,-4566.5275
C00488=36.693,-93.020,26.395,-179.9979,0.0053,-4568.4726
C00489=33.476,-94.189,26.358,179.9972,0.0435,-4570.4341
C00490=30.093,-95.074,26.301,179.9821,-0.1326,-4572.4363
C00491=26.720,-95.323,26.245,-179.7166,0.9262,-4574.3413
C00492=23.861,-94.948,26.175,-178.6786,2.3162,-4575.8934
C00493=21.871,-94.037,26.043,-176.8157,3.0731,-4576.9070
C00494=20.265,-92.865,25.771,-173.6100,5.1205,-4577.6899
C00495=18.686,-91.772,25.406,-169.1360,11.0995,-4578.4911
C00496=16.781,-91.008,25.041,-167.9432,21.7872,-4579.5526
C00497=13.981,-90.755,24.767,-174.6081,29.9498,-4581.2423
C00498=9.690,-91.047,24.657,-179.1672,31.6940,-4583.9250
C00499=5.020,-91.408,24.652,179.9386,31.7913,-4586.8566
C00500=0.000,-91.548,24.655,-180.0000,31.7764,-4590.0000
C00501=-5.020,-91.408,24.652,-179.9386,31.7913,-4593.1434
C00502=-9.690,-91.047,24.657,179.1672,31.6940,-4596.0750
C00503=-13.981,-90.755,24.767,174.6081,29.9498,-4598.7577
C00504=-16.781,-91.008,25.041,167.9432,21.7872,-4600.4474
C00505=-18.686,-91.772,25.406,169.1360,11.0995,-4601.5089
C00506=-20.265,-92.865,25.771,173.6100,5.1205,-4602.3101
C00507=-21.871,-94.037,26.043,176.8157,3.0731,-4603.0930
C00508=-23.861,-94.948,26.175,178.6786,2.3162,-4604.1066
C00509=-26.720,-95.323,26.245,179.7166,0.9262,-4605.6587
C00510=-30.093,-95.074,26.301,-179.9821,-0.1326,-4607.5637
C00511=-33.476,-94.189,26.358,-179.9972,0.0435,-4609.5659
C00512=-36.693,-93.020,26.395,179.9979,0.0053,-4611.5274
C00513=-39.829,-91.721,26.395,179.9977,0.0053,-4613.4725
C00514=-42.931,-90.273,26.358,179.9983,0.0436,-4615.4343
C00515=-45.948,-88.507,26.301,179.9790,-0.1336,-4617.4359
C00516=-48.509,-86.297,26.245,-179.7191,0.9269,-4619.3411
C00517=-50.266,-84.010,26.175,-178.6733,2.3167,-4620.8935
C00518=-51.029,-81.959,26.043,-176.8139,3.0727,-4621.9071
C00519=-51.336,-79.995,25.771,-173.6111,5.1213,-4622.6899
C00520=-51.679,-78.105,25.406,-169.1359,11.0962,-4623.4910
C00521=-52.487,-76.218,25.041,-167.9434,21.7869,-4624.5530
C00522=-54.287,-74.059,24.767,-174.6079,29.9481,-4626.2423
C00523=-57.528,-71.231,24.657,-179.1658,31.6931,-4628.9252
C00524=-61.085,-68.184,24.652,179.9356,31.7887,-4631.8567
C00525=-64.734,-64.734,24.655,-180.0000,31.7790,-4635.0000
C00526=-68.184,-61.085,24.652,-179.9356,31.7887,-4638.1433
C00527=-71.231,-57.528,24.657,179.1658,31.6931,-4641.0748
C00528=-74.059,-54.287,24.767,174.6079,29.9481,-4643.7577
C00529=-76.218,-52.487,25.041,167.9434,21.7869,-4645.4470
C00530=-78.105,-51.679,25.406,169.1359,11.0962,-4646.5090
C00531=-79.995,-51.336,25.771,173.6111,5.1213,-4647.3101
C00532=-81.959,-51.029,26.043,176.8139,3.0727,-4648.0929
C00533=-84.010,-50.266,26.175,178.6733,2.3167,-4649.1065
C00534=-86.297,-48.509,26.245,179.7191,0.9269,-4650.6589
C00535=-88.507,-45.948,26.301,-179.9790,-0.1336,-4652.5641
C00536=-90.273,-42.931,26.358,-179.9983,0.0436,-4654.5657
C00537=-91.721,-39.829,26.395,-179.9977,0.0053,-4656.5275
C00538=-93.020,-36.693,26.395,-179.9979,0.0053,-4658.4726
C00539=-94.189,-33.476,26.358,179.9972,0.0435,-4660.4341
C00540=-95.074,-30.093,26.301,179.9821,-0.1326,-4662.4363
C00541=-95.323,-26.720,26.245,-179.7166,0.9262,-4664.3413
C00542=-94.948,-23.861,26.175,-178.6786,2.3162,-4665.8934
C00543=-94.037,-21.871,26.043,-176.8157,3.0731,-4666.9070
C00544=-92.865,-20.265,25.771,-173.6100,5.1205,-4667.6899
C00545=-91.772,-18.686,25.406,-169.1360,11.0995,-4668.4911
C00546=-91.008,-16.781,25.041,-167.9432,21.7872,-4669.5526
C00547=-90.755,-13.981,24.767,-174.6081,29.9498,-4671.2423
C00548=-91.047,-9.690,24.657,-179.1672,31.6940,-4673.9250
C00549=-91.408,-5.020,24.652,179.9386,31.7913,-4676.8566
C00550=-91.548,0.000,24.655,180.0000,31.7764,-4680.0000
C00551=-91.408,5.020,24.652,-179.9386,31.7913,-4683.1434
C00552=-91.047,9.690,24.657,179.1672,31.6940,-4686.0750
C00553=-90.755,13.981,24.767,174.6081,29.9498,-4688.7577
C00554=-91.008,16.781,25.041,167.9432,21.7872,-4690.4474
C00555=-91.772,18.686,25.406,169.1360,11.0995,-4691.5089
C00556=-92.865,20.265,25.771,173.6100,5.1205,-4692.3101
C00557=-94.037,21.871,26.043,176.8157,3.0731,-4693.0930
C00558=-94.948,23.861,26.175,178.6786,2.3162,-4694.1066
C00559=-95.323,26.720,26.245,179.7166,0.9262,-4695.6587
C00560=-95.074,30.093,26.301,-179.9821,-0.1326,-4697.5637
C00561=-94.189,33.476,26.358,-179.9972,0.0435,-4699.5659
C00562=-93.020,36.693,26.395,179.9979,0.0053,-4701.5274
C00563=-91.721,39.829,26.395,179.9977,0.0053,-4703.4725
C00564=-90.273,42.931,26.358,179.9983,0.0436,-4705.4343
C00565=-88.507,45.948,26.301,179.9790,-0.1336,-4707.4359
C00566=-86.297,48.509,26.245,-179.7191,0.9269,-4709.3411
C00567=-84.010,50.266,26.175,-178.6733,2.3167,-4710.8935
C00568=-81.959,51.029,26.043,-176.8139,3.0727,-4711.9071
C00569=-79.995,51.336,25.771,-173.6111,5.1213,-4712.6899
C00570=-78.105,51.679,25.406,-169.1359,11.0962,-4713.4910
C00571=-76.218,52.487,25.041,-167.9434,21.7869,-4714.5530
C00572=-74.059,54.287,24.767,-174.6079,29.9481,-4716.2423
C00573=-71.231,57.528,24.657,-179.1658,31.6931,-4718.9252
C00574=-68.184,61.085,24.652,179.9356,31.7887,-4721.8567
C00575=-64.734,64.734,24.655,180.0000,31.7790,-4725.0000
C00576=-61.085,68.184,24.652,-179.9356,31.7887,-4728.1433
C00577=-57.528,71.231,24.657,179.1658,31.6931,-4731.0748
C00578=-54.287,74.059,24.767,174.6079,29.9481,-4733.7577
C00579=-52.487,76.218,25.041,167.9434,21.7869,-4735.4470
C00580=-51.679,78.105,25.406,169.1359,11.0962,-4736.5090
C00581=-51.336,79.995,25.771,173.6111,5.1213,-4737.3101
C00582=-51.029,81.959,26.043,176.8139,3.0727,-4738.0929
C00583=-50.266,84.010,26.175,178.6733,2.3167,-4739.1065
C00584=-48.509,86.297,26.245,179.7191,0.9269,-4740.6589
C00585=-45.948,88.507,26.301,-179.9790,-0.1336,-4742.5641
C00586=-42.931,90.273,26.358,-179.9983,0.0436,-4744.5657
C00587=-39.829,91.721,26.395,-179.9977,0.0053,-4746.5275
C00588=-36.693,93.020,26.395,-179.9979,0.0053,-4748.4726
C00589=-33.476,94.189,26.358,179.9972,0.0435,-4750.4341
C00590=-30.093,95.074,26.301,179.9821,-0.1326,-4752.4363
C00591=-26.720,95.323,26.245,-179.7166,0.9262,-4754.3413
C00592=-23.861,94.948,26.175,-178.6786,2.3162,-4755.8934
C00593=-21.871,94.037,26.043,-176.8157,3.0731,-4756.9070
C00594=-20.265,92.865,25.771,-173.6100,5.1205,-4757.6899
C00595=-18.686,91.772,25.406,-169.1360,11.0995,-4758.4911
C00596=-16.781,91.008,25.041,-167.9432,21.7872,-4759.5526
C00597=-13.981,90.755,24.767,-174.6081,29.9498,-4761.2423
C00598=-9.690,91.047,24.657,-179.1672,31.6940,-4763.9250
C00599=-5.020,91.408,24.652,179.9386,31.7913,-4766.8566
C00600=0.000,90.369,26.513,-180.0000,33.0099,-4770.0000
C00601=4.912,90.233,26.509,-179.9262,33.0210,-4773.1159
C00602=9.508,89.882,26.515,178.9946,32.9112,-4776.0385
C00603=13.759,89.629,26.645,173.5375,30.8885,-4778.7274
C00604=16.509,89.983,26.968,166.4353,20.8945,-4780.3963
C00605=18.373,90.901,27.402,169.1303,9.3354,-4781.4267
C00606=19.923,92.196,27.838,174.3403,3.7616,-4782.1938
C00607=21.502,93.597,28.166,177.5283,1.9745,-4782.9380
C00608=23.458,94.728,28.327,178.9719,1.5285,-4783.9087
C00609=26.340,95.277,28.411,179.8126,0.5486,-4785.4538
C00610=29.791,95.129,28.479,-179.9530,-0.3035,-4787.3887
C00611=33.285,94.252,28.548,-179.9987,0.0308,-4789.4506
C00612=36.628,93.045,28.594,-180.0000,0.0000,-4791.4875
C00613=39.893,91.693,28.594,-180.0000,0.0000,-4793.5125
C00614=43.110,90.182,28.548,179.9980,0.0308,-4795.5494
C00615=46.201,88.332,28.479,179.9517,-0.3033,-4797.6113
C00616=48.746,85.996,28.411,-179.8105,0.5487,-4799.5463
C00617=50.396,83.570,28.327,-178.9712,1.5238,-4801.0916
C00618=50.979,81.387,28.166,-177.5285,1.9748,-4802.0621
C00619=51.105,79.281,27.838,-174.3410,3.7642,-4802.8061
C00620=51.285,77.269,27.402,-169.1264,9.3352,-4803.5730
C00621=51.954,75.301,26.968,-166.4345,20.8949,-4804.6038
C00622=53.649,73.106,26.645,-173.5375,30.8897,-4806.2732
C00623=56.833,70.280,26.515,-178.9895,32.9101,-4808.9613
C00624=60.331,67.277,26.509,179.9267,33.0184,-4811.8843
C00625=63.901,63.901,26.513,-180.0000,33.0078,-4815.0000
C00626=67.277,60.331,26.509,-179.9267,33.0184,-4818.1157
C00627=70.280,56.833,26.515,178.9895,32.9101,-4821.0387
C00628=73.106,53.649,26.645,173.5375,30.8897,-4823.7268
C00629=75.301,51.954,26.968,166.4345,20.8949,-4825.3962
C00630=77.269,51.285,27.402,169.1264,9.3352,-4826.4270
C00631=79.281,51.105,27.838,174.3410,3.7642,-4827.1939
C00632=81.387,50.979,28.166,177.5285,1.9748,-4827.9379
C00633=83.570,50.396,28.327,178.9712,1.5238,-4828.9084
C00634=85.996,48.746,28.411,179.8105,0.5487,-4830.4537
C00635=88.332,46.201,28.479,-179.9517,-0.3033,-4832.3887
C00636=90.182,43.110,28.548,-179.9980,0.0308,-4834.4506
C00637=91.693,39.893,28.594,-180.0000,0.0000,-4836.4875
C00638=93.045,36.628,28.594,-180.0000,0.0000,-4838.5125
C00639=94.252,33.285,28.548,179.9987,0.0308,-4840.5494
C00640=95.129,29.791,28.479,179.9530,-0.3035,-4842.6113
C00641=95.277,26.340,28.411,-179.8126,0.5486,-4844.5462
C00642=94.728,23.458,28.327,-178.9719,1.5285,-4846.0913
C00643=93.597,21.502,28.166,-177.5283,1.9745,-4847.0620
C00644=92.196,19.923,27.838,-174.3403,3.7616,-4847.8062
C00645=90.901,18.373,27.402,-169.1303,9.3354,-4848.5733
C00646=89.983,16.509,26.968,-166.4353,20.8945,-4849.6037
C00647=89.629,13.759,26.645,-173.5375,30.8885,-4851.2726
C00648=89.882,9.508,26.515,-178.9946,32.9112,-4853.9615
C00649=90.233,4.912,26.509,179.9262,33.0210,-4856.8841
C00650=90.369,0.000,26.513,-180.0000,33.0099,-4860.0000
C00651=90.233,-4.912,26.509,-179.9262,33.0210,-4863.1159
C00652=89.882,-9.508,26.515,178.9946,32.9112,-4866.0385
C00653=89.629,-13.759,26.645,173.5375,30.8885,-4868.7274
C00654=89.983,-16.509,26.968,166.4353,20.8945,-4870.3963
C00655=90.901,-18.373,27.402,169.1303,9.3354,-4871.4267
C00656=92.196,-19.923,27.838,174.3403,3.7616,-4872.1938
C00657=93.597,-21.502,28.166,177.5283,1.9745,-4872.9380
C00658=94.728,-23.458,28.327,178.9719,1.5285,-4873.9087
C00659=95.277,-26.340,28.411,179.8126,0.5486,-4875.4538
C00660=95.129,-29.791,28.479,-179.9530,-0.3035,-4877.3887
C00661=94.252,-33.285,28.548,-179.9987,0.0308,-4879.4506
C00662=93.045,-36.628,28.594,-180.0000,0.0000,-4881.4875
C00663=91.693,-39.893,28.594,-180.0000,0.0000,-4883.5125
C00664=90.182,-43.110,28.548,179.9980,0.0308,-4885.5494
C00665=88.332,-46.201,28.479,179.9517,-0.3033,-4887.6113
C00666=85.996,-48.746,28.411,-179.8105,0.5487,-4889.5463
C00667=83.570,-50.396,28.327,-178.9712,1.5238,-4891.0916
C00668=81.387,-50.979,28.166,-177.5285,1.9748,-4892.0621
C00669=79.281,-51.105,27.838,-174.3410,3.7642,-4892.8061
C00670=77.269,-51.285,27.402,-169.1264,9.3352,-4893.5730
C00671=75.301,-51.954,26.968,-166.4345,20.8949,-4894.6038
C00672=73.106,-53.649,26.645,-173.5375,30.8897,-4896.2732
C00673=70.280,-56.833,26.515,-178.9895,32.9101,-4898.9613
C00674=67.277,-60.331,26.509,179.9267,33.0184,-4901.8843
C00675=63.901,-63.901,26.513,180.0000,33.0078,-4905.0000
C00676=60.331,-67.277,26.509,-179.9267,33.0184,-4908.1157
C00677=56.833,-70.280,26.515,178.9895,32.9101,-4911.0387
C00678=53.649,-73.106,26.645,173.5375,30.8897,-4913.7268
C00679=51.954,-75.301,26.968,166.4345,20.8949,-4915.3962
C00680=51.285,-77.269,27.402,169.1264,9.3352,-4916.4270
C00681=51.105,-79.281,27.838,174.3410,3.7642,-4917.1939
C00682=50.979,-81.387,28.166,177.5285,1.9748,-4917.9379
C00683=50.396,-83.570,28.327,178.9712,1.5238,-4918.9084
C00684=48.746,-85.996,28.411,179.8105,0.5487,-4920.4537
C00685=46.201,-88.332,28.479,-179.9517,-0.3033,-4922.3887
C00686=43.110,-90.182,28.548,-179.9980,0.0308,-4924.4506
C00687=39.893,-91.693,28.594,-180.0000,0.0000,-4926.4875
C00688=36.628,-93.045,28.594,-180.0000,0.0000,-4928.5125
C00689=33.285,-94.252,28.548,179.9987,0.0308,-4930.5494
C00690=29.791,-95.129,28.479,179.9530,-0.3035,-4932.6113
C00691=26.340,-95.277,28.411,-179.8126,0.5486,-4934.5462
C00692=23.458,-94.728,28.327,-178.9719,1.5285,-4936.0913
C00693=21.502,-93.597,28.166,-177.5283,1.9745,-4937.0620
C00694=19.923,-92.196,27.838,-174.3403,3.7616,-4937.8062
C00695=18.373,-90.901,27.402,-169.1303,9.3354,-4938.5733
C00696=16.509,-89.983,26.968,-166.4353,20.8945,-4939.6037
C00697=13.759,-89.629,26.645,-173.5375,30.8885,-4941.2726
C00698=9.508,-89.882,26.515,-178.9946,32.9112,-4943.9615
C00699=4.912,-90.233,26.509,179.9262,33.0210,-4946.8841
C00700=0.000,-90.369,26.513,180.0000,33.0099,-4950.0000
C00701=-4.912,-90.233,26.509,-179.9262,33.0210,-4953.1159
C00702=-9.508,-89.882,26.515,178.9946,32.9112,-4956.0385
C00703=-13.759,-89.629,26.645,173.5375,30.8885,-4958.7274
C00704=-16.509,-89.983,26.968,166.4353,20.8945,-4960.3963
C00705=-18.373,-90.901,27.402,169.1303,9.3354,-4961.4267
C00706=-19.923,-92.196,27.838,174.3403,3.7616,-4962.1938
C00707=-21.502,-93.597,28.166,177.5283,1.9745,-4962.9380
C00708=-23.458,-94.728,28.327,178.9719,1.5285,-4963.9087
C00709=-26.340,-95.277,28.411,179.8126,0.5486,-4965.4538
C00710=-29.791,-95.129,28.479,-179.9530,-0.3035,-4967.3887
C00711=-33.285,-94.252,28.548,-179.9987,0.0308,-4969.4506
C00712=-36.628,-93.045,28.594,-180.0000,0.0000,-4971.4875
C00713=-39.893,-91.693,28.594,-180.0000,0.0000,-4973.5125
C00714=-43.110,-90.182,28.548,179.9980,0.0308,-4975.5494
C00715=-46.201,-88.332,28.479,179.9517,-0.3033,-4977.6113
C00716=-48.746,-85.996,28.411,-179.8105,0.5487,-4979.5463
C00717=-50.396,-83.570,28.327,-178.9712,1.5238,-4981.0916
C00718=-50.979,-81.387,28.166,-177.5285,1.9748,-4982.0621
C00719=-51.105,-79.281,27.838,-174.3410,3.7642,-4982.8061
C00720=-51.285,-77.269,27.402,-169.1264,9.3352,-4983.5730
C00721=-51.954,-75.301,26.968,-166.4345,20.8949,-4984.6038
C00722=-53.649,-73.106,26.645,-173.5375,30.8897,-4986.2732
C00723=-56.833,-70.280,26.515,-178.9895,32.9101,-4988.9613
C00724=-60.331,-67.277,26.509,179.9267,33.0184,-4991.8843
C00725=-63.901,-63.901,26.513,-180.0000,33.0078,-4995.0000
C00726=-67.277,-60.331,26.509,-179.9267,33.0184,-4998.1157
C00727=-70.280,-56.833,26.515,178.9895,32.9101,-5001.0387
C00728=-73.106,-53.649,26.645,173.5375,30.8897,-5003.7268
C00729=-75.301,-51.954,26.968,166.4345,20.8949,-5005.3962
C00730=-77.269,-51.285,27.402,169.1264,9.3352,-5006.4270
C00731=-79.281,-51.105,27.838,174.3410,3.7642,-5007.1939
C00732=-81.387,-50.979,28.166,177.5285,1.9748,-5007.9379
C00733=-83.570,-50.396,28.327,178.9712,1.5238,-5008.9084
C00734=-85.996,-48.746,28.411,179.8105,0.5487,-5010.4537
C00735=-88.332,-46.201,28.479,-179.9517,-0.3033,-5012.3887
C00736=-90.182,-43.110,28.548,-179.9980,0.0308,-5014.4506
C00737=-91.693,-39.893,28.594,-180.0000,0.0000,-5016.4875
C00738=-93.045,-36.628,28.594,-180.0000,0.0000,-5018.5125
C00739=-94.252,-33.285,28.548,179.9987,0.0308,-5020.5494
C00740=-95.129,-29.791,28.479,179.9530,-0.3035,-5022.6113
C00741=-95.277,-26.340,28.411,-179.8126,0.5486,-5024.5462
C00742=-94.728,-23.458,28.327,-178.9719,1.5285,-5026.0913
C00743=-93.597,-21.502,28.166,-177.5283,1.9745,-5027.0620
C00744=-92.196,-19.923,27.838,-174.3403,3.7616,-5027.8062
C00745=-90.901,-18.373,27.402,-169.1303,9.3354,-5028.5733
C00746=-89.983,-16.509,26.968,-166.4353,20.8945,-5029.6037
C00747=-89.629,-13.759,26.645,-173.5375,30.8885,-5031.2726
C00748=-89.882,-9.508,26.515,-178.9946,32.9112,-5033.9615
C00749=-90.233,-4.912,26.509,179.9262,33.0210,-5036.8841
C00750=-90.369,0.000,26.513,-180.0000,33.0099,-5040.0000
C00751=-90.233,4.912,26.509,-179.9262,33.0210,-5043.1159
C00752=-89.882,9.508,26.515,178.9946,32.9112,-5046.0385
C00753=-89.629,13.759,26.645,173.5375,30.8885,-5048.7274
C00754=-89.983,16.509,26.968,166.4353,20.8945,-5050.3963
C00755=-90.901,18.373,27.402,169.1303,9.3354,-5051.4267
C00756=-92.196,19.923,27.838,174.3403,3.7616,-5052.1938
C00757=-93.597,21.502,28.166,177.5283,1.9745,-5052.9380
C00758=-94.728,23.458,28.327,178.9719,1.5285,-5053.9087
C00759=-95.277,26.340,28.411,179.8126,0.5486,-5055.4538
C00760=-95.129,29.791,28.479,-179.9530,-0.3035,-5057.3887
C00761=-94.252,33.285,28.548,-179.9987,0.0308,-5059.4506
C00762=-93.045,36.628,28.594,-180.0000,0.0000,-5061.4875
C00763=-91.693,39.893,28.594,-180.0000,0.0000,-5063.5125
C00764=-90.182,43.110,28.548,179.9980,0.0308,-5065.5494
C00765=-88.332,46.201,28.479,179.9517,-0.3033,-5067.6113
C00766=-85.996,48.746,28.411,-179.8105,0.5487,-5069.5463
C00767=-83.570,50.396,28.327,-178.9712,1.5238,-5071.0916
C00768=-81.387,50.979,28.166,-177.5285,1.9748,-5072.0621
C00769=-79.281,51.105,27.838,-174.3410,3.7642,-5072.8061
C00770=-77.269,51.285,27.402,-169.1264,9.3352,-5073.5730
C00771=-75.301,51.954,26.968,-166.4345,20.8949,-5074.6038
C00772=-73.106,53.649,26.645,-173.5375,30.8897,-5076.2732
C00773=-70.280,56.833,26.515,-178.9895,32.9101,-5078.9613
C00774=-67.277,60.331,26.509,179.9267,33.0184,-5081.8843
C00775=-63.901,63.901,26.513,-180.0000,33.0078,-5085.0000
C00776=-60.331,67.277,26.509,-179.9267,33.0184,-5088.1157
C00777=-56.833,70.280,26.515,178.9895,32.9101,-5091.0387
C00778=-53.649,73.106,26.645,173.5375,30.8897,-5093.7268
C00779=-51.954,75.301,26.968,166.4345,20.8949,-5095.3962
C00780=-51.285,77.269,27.402,169.1264,9.3352,-5096.4270
C00781=-51.105,79.281,27.838,174.3410,3.7642,-5097.1939
C00782=-50.979,81.387,28.166,177.5285,1.9748,-5097.9379
C00783=-50.396,83.570,28.327,178.9712,1.5238,-5098.9084
C00784=-48.746,85.996,28.411,179.8105,0.5487,-5100.4537
C00785=-46.201,88.332,28.479,-179.9517,-0.3033,-5102.3887
C00786=-43.110,90.182,28.548,-179.9980,0.0308,-5104.4506
C00787=-39.893,91.693,28.594,-180.0000,0.0000,-5106.4875
C00788=-36.628,93.045,28.594,-180.0000,0.0000,-5108.5125
C00789=-33.285,94.252,28.548,179.9987,0.0308,-5110.5494
C00790=-29.791,95.129,28.479,179.9530,-0.3035,-5112.6113
C00791=-26.340,95.277,28.411,-179.8126,0.5486,-5114.5462
C00792=-23.458,94.728,28.327,-178.9719,1.5285,-5116.0913
C00793=-21.502,93.597,28.166,-177.5283,1.9745,-5117.0620
C00794=-19.923,92.196,27.838,-174.3403,3.7616,-5117.8062
C00795=-18.373,90.901,27.402,-169.1303,9.3354,-5118.5733
C00796=-16.509,89.983,26.968,-166.4353,20.8945,-5119.6037
C00797=-13.759,89.629,26.645,-173.5375,30.8885,-5121.2726
C00798=-9.508,89.882,26.515,-178.9946,32.9112,-5123.9615
C00799=-4.912,90.233,26.509,179.9262,33.0210,-5126.8841
C00800=0.000,89.153,28.346,180.0000,34.0969,-5130.0000
C00801=4.801,89.020,28.341,-179.9168,34.1086,-5133.0871
C00802=9.321,88.681,28.348,178.8038,33.9818,-5136.0002
C00803=13.530,88.468,28.499,172.4066,31.6332,-5138.6952
C00804=16.227,88.922,28.874,165.2292,19.6025,-5140.3419
C00805=18.049,89.999,29.382,169.5475,7.5978,-5141.3400
C00806=19.567,91.502,29.895,175.3165,2.6020,-5142.0705
C00807=21.117,93.139,30.283,178.4639,1.0211,-5142.7745
C00808=23.038,94.499,30.474,179.4358,0.7176,-5143.7009
C00809=25.943,95.229,30.574,179.9458,0.1337,-5145.2391
C00810=29.476,95.186,30.656,-179.9144,-0.4893,-5147.2060
C00811=33.085,94.318,30.738,179.9997,0.0181,-5149.3299
C00812=36.560,93.071,30.793,-180.0000,0.0000,-5151.4458
C00813=39.959,91.663,30.793,-180.0000,0.0000,-5153.5540
C00814=43.298,90.088,30.738,-179.9998,0.0128,-5155.6698
C00815=46.464,88.150,30.656,179.9130,-0.4862,-5157.7938
C00816=48.993,85.682,30.574,-179.9460,0.1365,-5159.7609
C00817=50.531,83.111,30.474,-179.4372,0.7177,-5161.2994
C00818=50.927,80.791,30.283,-178.4682,1.0199,-5162.2255
C00819=50.865,78.538,29.895,-175.3211,2.6033,-5162.9290
C00820=50.876,76.401,29.382,-169.5498,7.5993,-5163.6599
C00821=51.403,74.351,28.874,-165.2308,19.5985,-5164.6583
C00822=52.989,72.123,28.499,-172.4037,31.6349,-5166.3048
C00823=56.115,69.298,28.348,-178.8001,33.9827,-5168.9993
C00824=59.552,66.342,28.341,179.9172,34.1079,-5171.9128
C00825=63.040,63.040,28.346,180.0000,34.0966,-5175.0000
C00826=66.342,59.552,28.341,-179.9172,34.1079,-5178.0872
C00827=69.298,56.115,28.348,178.8001,33.9827,-5181.0007
C00828=72.123,52.989,28.499,172.4037,31.6349,-5183.6952
C00829=74.351,51.403,28.874,165.2308,19.5985,-5185.3417
C00830=76.401,50.876,29.382,169.5498,7.5993,-5186.3401
C00831=78.538,50.865,29.895,175.3211,2.6033,-5187.0710
C00832=80.791,50.927,30.283,178.4682,1.0199,-5187.7745
C00833=83.111,50.531,30.474,179.4372,0.7177,-5188.7006
C00834=85.682,48.993,30.574,179.9460,0.1365,-5190.2391
C00835=88.150,46.464,30.656,-179.9130,-0.4862,-5192.2062
C00836=90.088,43.298,30.738,179.9998,0.0128,-5194.3302
C00837=91.663,39.959,30.793,-180.0000,0.0000,-5196.4460
C00838=93.071,36.560,30.793,-180.0000,0.0000,-5198.5542
C00839=94.318,33.085,30.738,-179.9997,0.0181,-5200.6701
C00840=95.186,29.476,30.656,179.9144,-0.4893,-5202.7940
C00841=95.229,25.943,30.574,-179.9458,0.1337,-5204.7609
C00842=94.499,23.038,30.474,-179.4358,0.7176,-5206.2991
C00843=93.139,21.117,30.283,-178.4639,1.0211,-5207.2255
C00844=91.502,19.567,29.895,-175.3165,2.6020,-5207.9295
C00845=89.999,18.049,29.382,-169.5475,7.5978,-5208.6600
C00846=88.922,16.227,28.874,-165.2292,19.6025,-5209.6581
C00847=88.468,13.530,28.499,-172.4066,31.6332,-5211.3048
C00848=88.681,9.321,28.348,-178.8038,33.9818,-5213.9998
C00849=89.020,4.801,28.341,179.9168,34.1086,-5216.9129
C00850=89.153,0.000,28.346,180.0000,34.0969,-5220.0000
C00851=89.020,-4.801,28.341,-179.9168,34.1086,-5223.0871
C00852=88.681,-9.321,28.348,178.8038,33.9818,-5226.0002
C00853=88.468,-13.530,28.499,172.4066,31.6332,-5228.6952
C00854=88.922,-16.227,28.874,165.2292,19.6025,-5230.3419
C00855=89.999,-18.049,29.382,169.5475,7.5978,-5231.3400
C00856=91.502,-19.567,29.895,175.3165,2.6020,-5232.0705
C00857=93.139,-21.117,30.283,178.4639,1.0211,-5232.7745
C00858=94.499,-23.038,30.474,179.4358,0.7176,-5233.7009
C00859=95.229,-25.943,30.574,179.9458,0.1337,-5235.2391
C00860=95.186,-29.476,30.656,-179.9144,-0.4893,-5237.2060
C00861=94.318,-33.085,30.738,179.9997,0.0181,-5239.3299
C00862=93.071,-36.560,30.793,-180.0000,0.0000,-5241.4458
C00863=91.663,-39.959,30.793,-180.0000,0.0000,-5243.5540
C00864=90.088,-43.298,30.738,-179.9998,0.0128,-5245.6698
C00865=88.150,-46.464,30.656,179.9130,-0.4862,-5247.7938
C00866=85.682,-48.993,30.574,-179.9460,0.1365,-5249.7609
C00867=83.111,-50.531,30.474,-179.4372,0.7177,-5251.2994
C00868=80.791,-50.927,30.283,-178.4682,1.0199,-5252.2255
C00869=78.538,-50.865,29.895,-175.3211,2.6033,-5252.9290
C00870=76.401,-50.876,29.382,-169.5498,7.5993,-5253.6599
C00871=74.351,-51.403,28.874,-165.2308,19.5985,-5254.6583
C00872=72.123,-52.989,28.499,-172.4037,31.6349,-5256.3048
C00873=69.298,-56.115,28.348,-178.8001,33.9827,-5258.9993
C00874=66.342,-59.552,28.341,179.9172,34.1079,-5261.9128
C00875=63.040,-63.040,28.346,-180.0000,34.0966,-5265.0000
C00876=59.552,-66.342,28.341,-179.9172,34.1079,-5268.0872
C00877=56.115,-69.298,28.348,178.8001,33.9827,-5271.0007
C00878=52.989,-72.123,28.499,172.4037,31.6349,-5273.6952
C00879=51.403,-74.351,28.874,165.2308,19.5985,-5275.3417
C00880=50.876,-76.401,29.382,169.5498,7.5993,-5276.3401
C00881=50.865,-78.538,29.895,175.3211,2.6033,-5277.0710
C00882=50.927,-80.791,30.283,178.4682,1.0199,-5277.7745
C00883=50.531,-83.111,30.474,179.4372,0.7177,-5278.7006
C00884=48.993,-85.682,30.574,179.9460,0.1365,-5280.2391
C00885=46.464,-88.150,30.656,-179.9130,-0.4862,-5282.2062
C00886=43.298,-90.088,30.738,179.9998,0.0128,-5284.3302
C00887=39.959,-91.663,30.793,-180.0000,0.0000,-5286.4460
C00888=36.560,-93.071,30.793,-180.0000,0.0000,-5288.5542
C00889=33.085,-94.318,30.738,-179.9997,0.0181,-5290.6701
C00890=29.476,-95.186,30.656,179.9144,-0.4893,-5292.7940
C00891=25.943,-95.229,30.574,-179.9458,0.1337,-5294.7609
C00892=23.038,-94.499,30.474,-179.4358,0.7176,-5296.2991
C00893=21.117,-93.139,30.283,-178.4639,1.0211,-5297.2255
C00894=19.567,-91.502,29.895,-175.3165,2.6020,-5297.9295
C00895=18.049,-89.999,29.382,-169.5475,7.5978,-5298.6600
C00896=16.227,-88.922,28.874,-165.2292,19.6025,-5299.6581
C00897=13.530,-88.468,28.499,-172.4066,31.6332,-5301.3048
C00898=9.321,-88.681,28.348,-178.8038,33.9818,-5303.9998
C00899=4.801,-89.020,28.341,179.9168,34.1086,-5306.9129
C00900=0.000,-89.153,28.346,-180.0000,34.0969,-5310.0000
C00901=-4.801,-89.020,28.341,-179.9168,34.1086,-5313.0871
C00902=-9.321,-88.681,28.348,178.8038,33.9818,-5316.0002
C00903=-13.530,-88.468,28.499,172.4066,31.6332,-5318.6952
C00904=-16.227,-88.922,28.874,165.2292,19.6025,-5320.3419
C00905=-18.049,-89.999,29.382,169.5475,7.5978,-5321.3400
C00906=-19.567,-91.502,29.895,175.3165,2.6020,-5322.0705
C00907=-21.117,-93.139,30.283,178.4639,1.0211,-5322.7745
C00908=-23.038,-94.499,30.474,179.4358,0.7176,-5323.7009
C00909=-25.943,-95.229,30.574,179.9458,0.1337,-5325.2391
C00910=-29.476,-95.186,30.656,-179.9144,-0.4893,-5327.2060
C00911=-33.085,-94.318,30.738,179.9997,0.0181,-5329.3299
C00912=-36.560,-93.071,30.793,-180.0000,0.0000,-5331.4458
C00913=-39.959,-91.663,30.793,-180.0000,0.0000,-5333.5540
C00914=-43.298,-90.088,30.738,-179.9998,0.0128,-5335.6698
C00915=-46.464,-88.150,30.656,179.9130,-0.4862,-5337.7938
C00916=-48.993,-85.682,30.574,-179.9460,0.1365,-5339.7609
C00917=-50.531,-83.111,30.474,-179.4372,0.7177,-5341.2994
C00918=-50.927,-80.791,30.283,-178.4682,1.0199,-5342.2255
C00919=-50.865,-78.538,29.895,-175.3211,2.6033,-5342.9290
C00920=-50.876,-76.401,29.382,-169.5498,7.5993,-5343.6599
C00921=-51.403,-74.351,28.874,-165.2308,19.5985,-5344.6583
C00922=-52.989,-72.123,28.499,-172.4037,31.6349,-5346.3048
C00923=-56.115,-69.298,28.348,-178.8001,33.9827,-5348.9993
C00924=-59.552,-66.342,28.341,179.9172,34.1079,-5351.9128
C00925=-63.040,-63.040,28.346,-180.0000,34.0966,-5355.0000
C00926=-66.342,-59.552,28.341,-179.9172,34.1079,-5358.0872
C00927=-69.298,-56.115,28.348,178.8001,33.9827,-5361.0007
C00928=-72.123,-52.989,28.499,172.4037,31.6349,-5363.6952
C00929=-74.351,-51.403,28.874,165.2308,19.5985,-5365.3417
C00930=-76.401,-50.876,29.382,169.5498,7.5993,-5366.3401
C00931=-78.538,-50.865,29.895,175.3211,2.6033,-5367.0710
C00932=-80.791,-50.927,30.283,178.4682,1.0199,-5367.7745
C00933=-83.111,-50.531,30.474,179.4372,0.7177,-5368.7006
C00934=-85.682,-48.993,30.574,179.9460,0.1365,-5370.2391
C00935=-88.150,-46.464,30.656,-179.9130,-0.4862,-5372.2062
C00936=-90.088,-43.298,30.738,179.9998,0.0128,-5374.3302
C00937=-91.663,-39.959,30.793,-180.0000,0.0000,-5376.4460
C00938=-93.071,-36.560,30.793,-180.0000,0.0000,-5378.5542
C00939=-94.318,-33.085,30.738,-179.9997,0.0181,-5380.6701
C00940=-95.186,-29.476,30.656,179.9144,-0.4893,-5382.7940
C00941=-95.229,-25.943,30.574,-179.9458,0.1337,-5384.7609
C00942=-94.499,-23.038,30.474,-179.4358,0.7176,-5386.2991
C00943=-93.139,-21.117,30.283,-178.4639,1.0211,-5387.2255
C00944=-91.502,-19.567,29.895,-175.3165,2.6020,-5387.9295
C00945=-89.999,-18.049,29.382,-169.5475,7.5978,-5388.6600
C00946=-88.922,-16.227,28.874,-165.2292,19.6025,-5389.6581
C00947=-88.468,-13.530,28.499,-172.4066,31.6332,-5391.3048
C00948=-88.681,-9.321,28.348,-178.8038,33.9818,-5393.9998
C00949=-89.020,-4.801,28.341,179.9168,34.1086,-5396.9129
C00950=-89.153,0.000,28.346,180.0000,34.0969,-5400.0000
C00951=-89.020,4.801,28.341,-179.9168,34.1086,-5403.0871
C00952=-88.681,9.321,28.348,178.8038,33.9818,-5406.0002
C00953=-88.468,13.530,28.499,172.4066,31.6332,-5408.6952
C00954=-88.922,16.227,28.874,165.2292,19.6025,-5410.3419
C00955=-89.999,18.049,29.382,169.5475,7.5978,-5411.3400
C00956=-91.502,19.567,29.895,175.3165,2.6020,-5412.0705
C00957=-93.139,21.117,30.283,178.4639,1.0211,-5412.7745
C00958=-94.499,23.038,30.474,179.4358,0.7176,-5413.7009
C00959=-95.229,25.943,30.574,179.9458,0.1337,-5415.2391
C00960=-95.186,29.476,30.656,-179.9144,-0.4893,-5417.2060
C00961=-94.318,33.085,30.738,179.9997,0.0181,-5419.3299
C00962=-93.071,36.560,30.793,-180.0000,0.0000,-5421.4458
C00963=-91.663,39.959,30.793,-180.0000,0.0000,-5423.5540
C00964=-90.088,43.298,30.738,-179.9998,0.0128,-5425.6698
C00965=-88.150,46.464,30.656,179.9130,-0.4862,-5427.7938
C00966=-85.682,48.993,30.574,-179.9460,0.1365,-5429.7609
C00967=-83.111,50.531,30.474,-179.4372,0.7177,-5431.2994
C00968=-80.791,50.927,30.283,-178.4682,1.0199,-5432.2255
C00969=-78.538,50.865,29.895,-175.3211,2.6033,-5432.9290
C00970=-76.401,50.876,29.382,-169.5498,7.5993,-5433.6599
C00971=-74.351,51.403,28.874,-165.2308,19.5985,-5434.6583
C00972=-72.123,52.989,28.499,-172.4037,31.6349,-5436.3048
C00973=-69.298,56.115,28.348,-178.8001,33.9827,-5438.9993
C00974=-66.342,59.552,28.341,179.9172,34.1079,-5441.9128
C00975=-63.040,63.040,28.346,180.0000,34.0966,-5445.0000
C00976=-59.552,66.342,28.341,-179.9172,34.1079,-5448.0872
C00977=-56.115,69.298,28.348,178.8001,33.9827,-5451.0007
C00978=-52.989,72.123,28.499,172.4037,31.6349,-5453.6952
C00979=-51.403,74.351,28.874,165.2308,19.5985,-5455.3417
C00980=-50.876,76.401,29.382,169.5498,7.5993,-5456.3401
C00981=-50.865,78.538,29.895,175.3211,2.6033,-5457.0710
C00982=-50.927,80.791,30.283,178.4682,1.0199,-5457.7745
C00983=-50.531,83.111,30.474,179.4372,0.7177,-5458.7006
C00984=-48.993,85.682,30.574,179.9460,0.1365,-5460.2391
C00985=-46.464,88.150,30.656,-179.9130,-0.4862,-5462.2062
C00986=-43.298,90.088,30.738,179.9998,0.0128,-5464.3302
C00987=-39.959,91.663,30.793,-180.0000,0.0000,-5466.4460
C00988=-36.560,93.071,30.793,-180.0000,0.0000,-5468.5542
C00989=-33.085,94.318,30.738,-179.9997,0.0181,-5470.6701
C00990=-29.476,95.186,30.656,179.9144,-0.4893,-5472.7940
C00991=-25.943,95.229,30.574,-179.9458,0.1337,-5474.7609
C00992=-23.038,94.499,30.474,-179.4358,0.7176,-5476.2991
C00993=-21.117,93.139,30.283,-178.4639,1.0211,-5477.2255
C00994=-19.567,91.502,29.895,-175.3165,2.6020,-5477.9295
C00995=-18.049,89.999,29.382,-169.5475,7.5978,-5478.6600
C00996=-16.227,88.922,28.874,-165.2292,19.6025,-5479.6581
C00997=-13.530,88.468,28.499,-172.4066,31.6332,-5481.3048
C00998=-9.321,88.681,28.348,-178.8038,33.9818,-5483.9998
C00999=-4.801,89.020,28.341,179.9168,34.1086,-5486.9129
C01000=0.000,87.904,30.157,-180.0000,35.0568,-5490.0000
C01001=4.687,87.776,30.152,-179.8975,35.0693,-5493.0565
C01002=9.129,87.447,30.160,178.5994,34.9274,-5495.9598
C01003=13.294,87.274,30.332,171.2309,32.1963,-5498.6610
C01004=15.938,87.830,30.762,164.3960,17.9884,-5500.2852
C01005=17.714,89.068,31.347,170.3040,6.0027,-5501.2483
C01006=19.200,90.783,31.942,176.4290,1.6678,-5501.9417
C01007=20.718,92.664,32.394,179.5311,0.2592,-5502.6030
C01008=22.602,94.262,32.617,-179.9450,-0.0575,-5503.4837
C01009=25.531,95.180,32.735,-179.8726,-0.2980,-5505.0155
C01010=29.149,95.246,32.831,-179.8662,-0.6721,-5507.0162
C01011=32.878,94.386,32.928,-180.0000,-0.0000,-5509.2050
C01012=36.490,93.098,32.991,-180.0000,-0.0000,-5511.4028
C01013=40.028,91.633,32.991,-180.0000,-0.0000,-5513.5971
C01014=43.493,89.989,32.928,-180.0000,-0.0000,-5515.7952
C01015=46.737,87.960,32.831,179.8655,-0.6749,-5517.9837
C01016=49.249,85.356,32.735,179.8712,-0.2926,-5519.9842
C01017=50.671,82.635,32.617,179.9485,-0.0585,-5521.5162
C01018=50.874,80.174,32.394,-179.5347,0.2613,-5522.3970
C01019=50.617,77.770,31.942,-176.4306,1.6678,-5523.0583
C01020=50.455,75.506,31.347,-170.3014,6.0013,-5523.7518
C01021=50.836,73.375,30.762,-164.3944,17.9871,-5524.7152
C01022=52.312,71.113,30.332,-171.2278,32.1987,-5526.3389
C01023=55.379,68.290,30.160,-178.5955,34.9311,-5529.0399
C01024=58.753,65.381,30.152,179.9021,35.0679,-5531.9437
C01025=62.157,62.157,30.157,-179.9951,35.0560,-5535.0000
C01026=65.381,58.753,30.152,-179.9021,35.0679,-5538.0563
C01027=68.290,55.379,30.160,178.5911,34.9274,-5540.9601
C01028=71.113,52.312,30.332,171.2332,32.1958,-5543.6611
C01029=73.375,50.836,30.762,164.3944,17.9871,-5545.2848
C01030=75.506,50.455,31.347,170.3014,6.0013,-5546.2482
C01031=77.770,50.617,31.942,176.4306,1.6678,-5546.9417
C01032=80.174,50.874,32.394,179.5347,0.2613,-5547.6030
C01033=82.635,50.671,32.617,-179.9485,-0.0585,-5548.4838
C01034=85.356,49.249,32.735,-179.8712,-0.2926,-5550.0158
C01035=87.960,46.737,32.831,-179.8655,-0.6749,-5552.0163
C01036=89.989,43.493,32.928,-180.0000,-0.0000,-5554.2048
C01037=91.633,40.028,32.991,-180.0000,-0.0000,-5556.4029
C01038=93.098,36.490,32.991,-180.0000,-0.0000,-5558.5972
C01039=94.386,32.878,32.928,-180.0000,-0.0000,-5560.7950
C01040=95.246,29.149,32.831,179.8662,-0.6721,-5562.9838
C01041=95.180,25.531,32.735,179.8726,-0.2980,-5564.9845
C01042=94.262,22.602,32.617,179.9450,-0.0575,-5566.5163
C01043=92.664,20.718,32.394,-179.5311,0.2592,-5567.3970
C01044=90.783,19.200,31.942,-176.4290,1.6678,-5568.0583
C01045=89.068,17.714,31.347,-170.3040,6.0027,-5568.7517
C01046=87.830,15.938,30.762,-164.3960,17.9884,-5569.7148
C01047=87.274,13.294,30.332,-171.2309,32.1963,-5571.3390
C01048=87.447,9.129,30.160,-178.5994,34.9274,-5574.0402
C01049=87.776,4.687,30.152,179.8975,35.0693,-5576.9435
C01050=87.904,0.000,30.157,-180.0000,35.0568,-5580.0000
C01051=87.776,-4.687,30.152,-179.9045,35.0690,-5583.0565
C01052=87.447,-9.130,30.160,178.5920,34.9269,-5585.9604
C01053=87.274,-13.294,30.332,171.2309,32.1963,-5588.6610
C01054=87.830,-15.938,30.762,164.3960,17.9884,-5590.2852
C01055=89.068,-17.714,31.347,170.3040,6.0027,-5591.2483
C01056=90.783,-19.200,31.942,176.4290,1.6678,-5591.9417
C01057=92.664,-20.718,32.394,179.5311,0.2592,-5592.6030
C01058=94.262,-22.602,32.617,-179.9450,-0.0575,-5593.4837
C01059=95.180,-25.531,32.735,-179.8726,-0.2980,-5595.0155
C01060=95.246,-29.149,32.831,-179.8662,-0.6721,-5597.0162
C01061=94.386,-32.878,32.928,-180.0000,-0.0000,-5599.2050
C01062=93.098,-36.490,32.991,-180.0000,-0.0000,-5601.4028
C01063=91.633,-40.028,32.991,-180.0000,-0.0000,-5603.5971
C01064=89.989,-43.493,32.928,-180.0000,-0.0000,-5605.7952
C01065=87.960,-46.737,32.831,179.8655,-0.6749,-5607.9837
C01066=85.356,-49.249,32.735,179.8712,-0.2926,-5609.9842
C01067=82.635,-50.671,32.617,179.9485,-0.0585,-5611.5162
C01068=80.174,-50.874,32.394,-179.5347,0.2613,-5612.3970
C01069=77.770,-50.617,31.942,-176.4306,1.6678,-5613.0583
C01070=75.506,-50.455,31.347,-170.3014,6.0013,-5613.7518
C01071=73.375,-50.836,30.762,-164.3944,17.9871,-5614.7152
C01072=71.113,-52.312,30.332,-171.2278,32.1987,-5616.3389
C01073=68.290,-55.379,30.160,-178.5955,34.9311,-5619.0399
C01074=65.381,-58.753,30.152,179.9021,35.0679,-5621.9437
C01075=62.157,-62.157,30.157,-179.9951,35.0560,-5625.0000
C01076=58.753,-65.381,30.152,-179.9021,35.0679,-5628.0563
C01077=55.379,-68.290,30.160,178.5911,34.9274,-5630.9601
C01078=52.312,-71.113,30.332,171.2332,32.1958,-5633.6611
C01079=50.836,-73.375,30.762,164.3944,17.9871,-5635.2848
C01080=50.455,-75.506,31.347,170.3014,6.0013,-5636.2482
C01081=50.617,-77.770,31.942,176.4306,1.6678,-5636.9417
C01082=50.874,-80.174,32.394,179.5347,0.2613,-5637.6030
C01083=50.671,-82.635,32.617,-179.9485,-0.0585,-5638.4838
C01084=49.249,-85.356,32.735,-179.8712,-0.2926,-5640.0158
C01085=46.737,-87.960,32.831,-179.8655,-0.6749,-5642.0163
C01086=43.493,-89.989,32.928,-180.0000,-0.0000,-5644.2048
C01087=40.028,-91.633,32.991,-180.0000,-0.0000,-5646.4029
C01088=36.490,-93.098,32.991,-180.0000,-0.0000,-5648.5972
C01089=32.878,-94.386,32.928,-180.0000,-0.0000,-5650.7950
C01090=29.149,-95.246,32.831,179.8662,-0.6721,-5652.9838
C01091=25.531,-95.180,32.735,179.8726,-0.2980,-5654.9845
C01092=22.602,-94.262,32.617,179.9450,-0.0575,-5656.5163
C01093=20.718,-92.664,32.394,-179.5311,0.2592,-5657.3970
C01094=19.200,-90.783,31.942,-176.4290,1.6678,-5658.0583
C01095=17.714,-89.068,31.347,-170.3040,6.0027,-5658.7517
C01096=15.938,-87.830,30.762,-164.3960,17.9884,-5659.7148
C01097=13.294,-87.274,30.332,-171.2309,32.1963,-5661.3390
C01098=9.129,-87.447,30.160,-178.5994,34.9274,-5664.0402
C01099=4.687,-87.776,30.152,179.8975,35.0693,-5666.9435
C01100=0.000,-87.904,30.157,180.0000,35.0568,-5670.0000
C01101=-4.687,-87.776,30.152,-179.9045,35.0690,-5673.0565
C01102=-9.130,-87.447,30.160,178.5920,34.9269,-5675.9604
C01103=-13.294,-87.274,30.332,171.2309,32.1963,-5678.6610
C01104=-15.938,-87.830,30.762,164.3960,17.9884,-5680.2852
C01105=-17.714,-89.068,31.347,170.3040,6.0027,-5681.2483
C01106=-19.200,-90.783,31.942,176.4290,1.6678,-5681.9417
C01107=-20.718,-92.664,32.394,179.5311,0.2592,-5682.6030
C01108=-22.602,-94.262,32.617,-179.9450,-0.0575,-5683.4837
C01109=-25.531,-95.180,32.735,-179.8726,-0.2980,-5685.0155
C01110=-29.149,-95.246,32.831,-179.8662,-0.6721,-5687.0162
C01111=-32.878,-94.386,32.928,-180.0000,-0.0000,-5689.2050
C01112=-36.490,-93.098,32.991,-180.0000,-0.0000,-5691.4028
C01113=-40.028,-91.633,32.991,-180.0000,-0.0000,-5693.5971
C01114=-43.493,-89.989,32.928,-180.0000,-0.0000,-5695.7952
C01115=-46.737,-87.960,32.831,179.8655,-0.6749,-5697.9837
C01116=-49.249,-85.356,32.735,179.8712,-0.2926,-5699.9842
C01117=-50.671,-82.635,32.617,179.9485,-0.0585,-5701.5162
C01118=-50.874,-80.174,32.394,-179.5347,0.2613,-5702.3970
C01119=-50.617,-77.770,31.942,-176.4306,1.6678,-5703.0583
C01120=-50.455,-75.506,31.347,-170.3014,6.0013,-5703.7518
C01121=-50.836,-73.375,30.762,-164.3944,17.9871,-5704.7152
C01122=-52.312,-71.113,30.332,-171.2278,32.1987,-5706.3389
C01123=-55.379,-68.290,30.160,-178.5955,34.9311,-5709.0399
C01124=-58.753,-65.381,30.152,179.9021,35.0679,-5711.9437
C01125=-62.157,-62.157,30.157,-179.9951,35.0560,-5715.0000
C01126=-65.381,-58.753,30.152,-179.9021,35.0679,-5718.0563
C01127=-68.290,-55.379,30.160,178.5911,34.9274,-5720.9601
C01128=-71.113,-52.312,30.332,171.2332,32.1958,-5723.6611
C01129=-73.375,-50.836,30.762,164.3944,17.9871,-5725.2848
C01130=-75.506,-50.455,31.347,170.3014,6.0013,-5726.2482
C01131=-77.770,-50.617,31.942,176.4306,1.6678,-5726.9417
C01132=-80.174,-50.874,32.394,179.5347,0.2613,-5727.6030
C01133=-82.635,-50.671,32.617,-179.9485,-0.0585,-5728.4838
C01134=-85.356,-49.249,32.735,-179.8712,-0.2926,-5730.0158
C01135=-87.960,-46.737,32.831,-179.8655,-0.6749,-5732.0163
C01136=-89.989,-43.493,32.928,-180.0000,-0.0000,-5734.2048
C01137=-91.633,-40.028,32.991,-180.0000,-0.0000,-5736.4029
C01138=-93.098,-36.490,32.991,-180.0000,-0.0000,-5738.5972
C01139=-94.386,-32.878,32.928,-180.0000,-0.0000,-5740.7950
C01140=-95.246,-29.149,32.831,179.8662,-0.6721,-5742.9838
C01141=-95.180,-25.531,32.735,179.8726,-0.2980,-5744.9845
C01142=-94.262,-22.602,32.617,179.9450,-0.0575,-5746.5163
C01143=-92.664,-20.718,32.394,-179.5311,0.2592,-5747.3970
C01144=-90.783,-19.200,31.942,-176.4290,1.6678,-5748.0583
C01145=-89.068,-17.714,31.347,-170.3040,6.0027,-5748.7517
C01146=-87.830,-15.938,30.762,-164.3960,17.9884,-5749.7148
C01147=-87.274,-13.294,30.332,-171.2309,32.1963,-5751.3390
C01148=-87.447,-9.129,30.160,-178.5994,34.9274,-5754.0402
C01149=-87.776,-4.687,30.152,179.8975,35.0693,-5756.9435
C01150=-87.904,0.000,30.157,-180.0000,35.0568,-5760.0000
C01151=-87.776,4.687,30.152,-179.9045,35.0690,-5763.0565
C01152=-87.447,9.130,30.160,178.5920,34.9269,-5765.9604
C01153=-87.274,13.294,30.332,171.2309,32.1963,-5768.6610
C01154=-87.830,15.938,30.762,164.3960,17.9884,-5770.2852
C01155=-89.068,17.714,31.347,170.3040,6.0027,-5771.2483
C01156=-90.783,19.200,31.942,176.4290,1.6678,-5771.9417
C01157=-92.664,20.718,32.394,179.5311,0.2592,-5772.6030
C01158=-94.262,22.602,32.617,-179.9450,-0.0575,-5773.4837
C01159=-95.180,25.531,32.735,-179.8726,-0.2980,-5775.0155
C01160=-95.246,29.149,32.831,-179.8662,-0.6721,-5777.0162
C01161=-94.386,32.878,32.928,-180.0000,-0.0000,-5779.2050
C01162=-93.098,36.490,32.991,-180.0000,-0.0000,-5781.4028
C01163=-91.633,40.028,32.991,-180.0000,-0.0000,-5783.5971
C01164=-89.989,43.493,32.928,-180.0000,-0.0000,-5785.7952
C01165=-87.960,46.737,32.831,179.8655,-0.6749,-5787.9837
C01166=-85.356,49.249,32.735,179.8712,-0.2926,-5789.9842
C01167=-82.635,50.671,32.617,179.9485,-0.0585,-5791.5162
C01168=-80.174,50.874,32.394,-179.5347,0.2613,-5792.3970
C01169=-77.770,50.617,31.942,-176.4306,1.6678,-5793.0583
C01170=-75.506,50.455,31.347,-170.3014,6.0013,-5793.7518
C01171=-73.375,50.836,30.762,-164.3944,17.9871,-5794.7152
C01172=-71.113,52.312,30.332,-171.2278,32.1987,-5796.3389
C01173=-68.290,55.379,30.160,-178.5955,34.9311,-5799.0399
C01174=-65.381,58.753,30.152,179.9021,35.0679,-5801.9437
C01175=-62.157,62.157,30.157,-179.9951,35.0560,-5805.0000
C01176=-58.753,65.381,30.152,-179.9021,35.0679,-5808.0563
C01177=-55.379,68.290,30.160,178.5911,34.9274,-5810.9601
C01178=-52.312,71.113,30.332,171.2332,32.1958,-5813.6611
C01179=-50.836,73.375,30.762,164.3944,17.9871,-5815.2848
C01180=-50.455,75.506,31.347,170.3014,6.0013,-5816.2482
C01181=-50.617,77.770,31.942,176.4306,1.6678,-5816.9417
C01182=-50.874,80.174,32.394,179.5347,0.2613,-5817.6030
C01183=-50.671,82.635,32.617,-179.9485,-0.0585,-5818.4838
C01184=-49.249,85.356,32.735,-179.8712,-0.2926,-5820.0158
C01185=-46.737,87.960,32.831,-179.8655,-0.6749,-5822.0163
C01186=-43.493,89.989,32.928,-180.0000,-0.0000,-5824.2048
C01187=-40.028,91.633,32.991,-180.0000,-0.0000,-5826.4029
C01188=-36.490,93.098,32.991,-180.0000,-0.0000,-5828.5972
C01189=-32.878,94.386,32.928,-180.0000,-0.0000,-5830.7950
C01190=-29.149,95.246,32.831,179.8662,-0.6721,-5832.9838
C01191=-25.531,95.180,32.735,179.8726,-0.2980,-5834.9845
C01192=-22.602,94.262,32.617,179.9450,-0.0575,-5836.5163
C01193=-20.718,92.664,32.394,-179.5311,0.2592,-5837.3970
C01194=-19.200,90.783,31.942,-176.4290,1.6678,-5838.0583
C01195=-17.714,89.068,31.347,-170.3040,6.0027,-5838.7517
C01196=-15.938,87.830,30.762,-164.3960,17.9884,-5839.7148
C01197=-13.294,87.274,30.332,-171.2309,32.1963,-5841.3390
C01198=-9.130,87.447,30.160,-178.5920,34.9269,-5844.0396
C01199=-4.687,87.776,30.152,179.9045,35.0690,-5846.9435
C01200=0.000,86.627,31.948,180.0000,35.8947,-5850.0000
C01201=4.570,86.503,31.943,-179.8896,35.9073,-5853.0242
C01202=8.933,86.186,31.951,178.3732,35.7506,-5855.9175
C01203=13.053,86.053,32.146,170.0298,32.5775,-5858.6252
C01204=15.641,86.712,32.633,163.9561,16.1560,-5860.2250
C01205=17.370,88.113,33.299,171.2911,4.6136,-5861.1519
C01206=18.822,90.045,33.980,177.5928,0.9554,-5861.8065
C01207=20.308,92.176,34.500,-179.3523,-0.3032,-5862.4248
C01208=22.152,94.017,34.757,-179.2110,-0.7502,-5863.2580
C01209=25.107,95.129,34.893,-179.6486,-0.7251,-5864.7847
C01210=28.812,95.307,35.004,-179.8159,-0.8662,-5866.8204
C01211=32.664,94.457,35.116,-179.9998,-0.0181,-5869.0758
C01212=36.417,93.126,35.190,-179.9979,-0.0053,-5871.3580
C01213=40.099,91.601,35.190,-179.9977,-0.0052,-5873.6417
C01214=43.694,89.888,35.116,-179.9976,-0.0180,-5875.9241
C01215=47.019,87.765,35.004,179.8142,-0.8665,-5878.1796
C01216=49.513,85.019,34.893,179.6485,-0.7285,-5880.2155
C01217=50.816,82.144,34.757,179.2111,-0.7508,-5881.7418
C01218=50.818,79.538,34.500,179.3519,-0.3053,-5882.5751
C01219=50.362,76.980,33.980,-177.5895,0.9541,-5883.1936
C01220=50.022,74.588,33.299,-171.2890,4.6171,-5883.8475
C01221=50.255,72.374,32.633,-163.9525,16.1553,-5884.7753
C01222=51.619,70.079,32.146,-170.0305,32.5797,-5886.3747
C01223=54.626,67.259,31.951,-178.3760,35.7490,-5889.0826
C01224=57.935,64.399,31.943,179.8882,35.9085,-5891.9754
C01225=61.254,61.254,31.948,180.0000,35.8962,-5895.0000
C01226=64.398,57.936,31.943,-179.8875,35.9085,-5898.0237
C01227=67.259,54.626,31.951,178.3760,35.7490,-5900.9174
C01228=70.079,51.619,32.146,170.0305,32.5797,-5903.6253
C01229=72.374,50.255,32.633,163.9525,16.1553,-5905.2247
C01230=74.588,50.022,33.299,171.2890,4.6171,-5906.1525
C01231=76.980,50.362,33.980,177.5895,0.9541,-5906.8064
C01232=79.538,50.818,34.500,-179.3519,-0.3053,-5907.4249
C01233=82.144,50.816,34.757,-179.2111,-0.7508,-5908.2582
C01234=85.019,49.513,34.893,-179.6485,-0.7285,-5909.7845
C01235=87.765,47.019,35.004,-179.8142,-0.8665,-5911.8204
C01236=89.888,43.694,35.116,179.9976,-0.0180,-5914.0759
C01237=91.601,40.099,35.190,179.9977,-0.0052,-5916.3583
C01238=93.126,36.417,35.190,179.9979,-0.0053,-5918.6420
C01239=94.457,32.664,35.116,179.9998,-0.0181,-5920.9242
C01240=95.307,28.812,35.004,179.8159,-0.8662,-5923.1796
C01241=95.129,25.107,34.893,179.6486,-0.7251,-5925.2153
C01242=94.017,22.152,34.757,179.2110,-0.7502,-5926.7420
C01243=92.176,20.308,34.500,179.3523,-0.3032,-5927.5752
C01244=90.045,18.822,33.980,-177.5928,0.9554,-5928.1935
C01245=88.113,17.370,33.299,-171.2911,4.6136,-5928.8481
C01246=86.712,15.641,32.633,-163.9561,16.1560,-5929.7750
C01247=86.053,13.053,32.146,-170.0298,32.5775,-5931.3748
C01248=86.186,8.933,31.951,-178.3732,35.7506,-5934.0825
C01249=86.503,4.570,31.943,179.8896,35.9073,-5936.9758
C01250=86.627,0.000,31.948,-180.0000,35.8947,-5940.0000
C01251=86.503,-4.570,31.943,-179.8896,35.9073,-5943.0242
C01252=86.186,-8.933,31.951,178.3732,35.7506,-5945.9175
C01253=86.053,-13.053,32.146,170.0298,32.5775,-5948.6252
C01254=86.712,-15.641,32.633,163.9561,16.1560,-5950.2250
C01255=88.113,-17.370,33.299,171.2911,4.6136,-5951.1519
C01256=90.045,-18.822,33.980,177.5928,0.9554,-5951.8065
C01257=92.176,-20.308,34.500,-179.3523,-0.3032,-5952.4248
C01258=94.017,-22.152,34.757,-179.2110,-0.7502,-5953.2580
C01259=95.129,-25.107,34.893,-179.6486,-0.7251,-5954.7847
C01260=95.307,-28.812,35.004,-179.8159,-0.8662,-5956.8204
C01261=94.457,-32.664,35.116,-179.9998,-0.0181,-5959.0758
C01262=93.126,-36.417,35.190,-179.9979,-0.0053,-5961.3580
C01263=91.601,-40.099,35.190,-179.9977,-0.0052,-5963.6417
C01264=89.888,-43.694,35.116,-179.9976,-0.0180,-5965.9241
C01265=87.765,-47.019,35.004,179.8142,-0.8665,-5968.1796
C01266=85.019,-49.513,34.893,179.6485,-0.7285,-5970.2155
C01267=82.144,-50.816,34.757,179.2111,-0.7508,-5971.7418
C01268=79.538,-50.818,34.500,179.3519,-0.3053,-5972.5751
C01269=76.980,-50.362,33.980,-177.5895,0.9541,-5973.1936
C01270=74.588,-50.022,33.299,-171.2890,4.6171,-5973.8475
C01271=72.374,-50.255,32.633,-163.9525,16.1553,-5974.7753
C01272=70.079,-51.619,32.146,-170.0305,32.5797,-5976.3747
C01273=67.259,-54.626,31.951,-178.3760,35.7490,-5979.0826
C01274=64.399,-57.935,31.943,179.8882,35.9085,-5981.9754
C01275=61.254,-61.254,31.948,-180.0000,35.8962,-5985.0000
C01276=57.936,-64.398,31.943,-179.8875,35.9085,-5988.0237
C01277=54.626,-67.259,31.951,178.3760,35.7490,-5990.9174
C01278=51.619,-70.079,32.146,170.0305,32.5797,-5993.6253
C01279=50.255,-72.374,32.633,163.9525,16.1553,-5995.2247
C01280=50.022,-74.588,33.299,171.2890,4.6171,-5996.1525
C01281=50.362,-76.980,33.980,177.5895,0.9541,-5996.8064
C01282=50.818,-79.538,34.500,-179.3519,-0.3053,-5997.4249
C01283=50.816,-82.144,34.757,-179.2111,-0.7508,-5998.2582
C01284=49.513,-85.019,34.893,-179.6485,-0.7285,-5999.7845
C01285=47.019,-87.765,35.004,-179.8142,-0.8665,-6001.8204
C01286=43.694,-89.888,35.116,179.9976,-0.0180,-6004.0759
C01287=40.099,-91.601,35.190,179.9977,-0.0052,-6006.3583
C01288=36.417,-93.126,35.190,179.9979,-0.0053,-6008.6420
C01289=32.664,-94.457,35.116,179.9998,-0.0181,-6010.9242
C01290=28.812,-95.307,35.004,179.8159,-0.8662,-6013.1796
C01291=25.107,-95.129,34.893,179.6486,-0.7251,-6015.2153
C01292=22.152,-94.017,34.757,179.2110,-0.7502,-6016.7420
C01293=20.308,-92.176,34.500,179.3523,-0.3032,-6017.5752
C01294=18.822,-90.045,33.980,-177.5928,0.9554,-6018.1935
C01295=17.370,-88.113,33.299,-171.2911,4.6136,-6018.8481
C01296=15.641,-86.712,32.633,-163.9561,16.1560,-6019.7750
C01297=13.053,-86.053,32.146,-170.0298,32.5775,-6021.3748
C01298=8.933,-86.186,31.951,-178.3732,35.7506,-6024.0825
C01299=4.570,-86.503,31.943,179.8896,35.9073,-6026.9758
C01300=0.000,-86.627,31.948,-180.0000,35.8947,-6030.0000
C01301=-4.570,-86.503,31.943,-179.8896,35.9073,-6033.0242
C01302=-8.933,-86.186,31.951,178.3732,35.7506,-6035.9175
C01303=-13.053,-86.053,32.146,170.0298,32.5775,-6038.6252
C01304=-15.641,-86.712,32.633,163.9561,16.1560,-6040.2250
C01305=-17.370,-88.113,33.299,171.2911,4.6136,-6041.1519
C01306=-18.822,-90.045,33.980,177.5928,0.9554,-6041.8065
C01307=-20.308,-92.176,34.500,-179.3523,-0.3032,-6042.4248
C01308=-22.152,-94.017,34.757,-179.2110,-0.7502,-6043.2580
C01309=-25.107,-95.129,34.893,-179.6486,-0.7251,-6044.7847
C01310=-28.812,-95.307,35.004,-179.8159,-0.8662,-6046.8204
C01311=-32.664,-94.457,35.116,-179.9998,-0.0181,-6049.0758
C01312=-36.417,-93.126,35.190,-179.9979,-0.0053,-6051.3580
C01313=-40.099,-91.601,35.190,-179.9977,-0.0052,-6053.6417
C01314=-43.694,-89.888,35.116,-179.9976,-0.0180,-6055.9241
C01315=-47.019,-87.765,35.004,179.8142,-0.8665,-6058.1796
C01316=-49.513,-85.019,34.893,179.6485,-0.7285,-6060.2155
C01317=-50.816,-82.144,34.757,179.2111,-0.7508,-6061.7418
C01318=-50.818,-79.538,34.500,179.3519,-0.3053,-6062.5751
C01319=-50.362,-76.980,33.980,-177.5895,0.9541,-6063.1936
C01320=-50.022,-74.588,33.299,-171.2890,4.6171,-6063.8475
C01321=-50.255,-72.374,32.633,-163.9525,16.1553,-6064.7753
C01322=-51.619,-70.079,32.146,-170.0305,32.5797,-6066.3747
C01323=-54.626,-67.259,31.951,-178.3760,35.7490,-6069.0826
C01324=-57.935,-64.399,31.943,179.8882,35.9085,-6071.9754
C01325=-61.254,-61.254,31.948,-180.0000,35.8962,-6075.0000
C01326=-64.398,-57.936,31.943,-179.8875,35.9085,-6078.0237
C01327=-67.259,-54.626,31.951,178.3760,35.7490,-6080.9174
C01328=-70.079,-51.619,32.146,170.0305,32.5797,-6083.6253
C01329=-72.374,-50.255,32.633,163.9525,16.1553,-6085.2247
C01330=-74.588,-50.022,33.299,171.2890,4.6171,-6086.1525
C01331=-76.980,-50.362,33.980,177.5895,0.9541,-6086.8064
C01332=-79.538,-50.818,34.500,-179.3519,-0.3053,-6087.4249
C01333=-82.144,-50.816,34.757,-179.2111,-0.7508,-6088.2582
C01334=-85.019,-49.513,34.893,-179.6485,-0.7285,-6089.7845
C01335=-87.765,-47.019,35.004,-179.8142,-0.8665,-6091.8204
C01336=-89.888,-43.694,35.116,179.9976,-0.0180,-6094.0759
C01337=-91.601,-40.099,35.190,179.9977,-0.0052,-6096.3583
C01338=-93.126,-36.417,35.190,179.9979,-0.0053,-6098.6420
C01339=-94.457,-32.664,35.116,179.9998,-0.0181,-6100.9242
C01340=-95.307,-28.812,35.004,179.8159,-0.8662,-6103.1796
C01341=-95.129,-25.107,34.893,179.6486,-0.7251,-6105.2153
C01342=-94.017,-22.152,34.757,179.2110,-0.7502,-6106.7420
C01343=-92.176,-20.308,34.500,179.3523,-0.3032,-6107.5752
C01344=-90.045,-18.822,33.980,-177.5928,0.9554,-6108.1935
C01345=-88.113,-17.370,33.299,-171.2911,4.6136,-6108.8481
C01346=-86.712,-15.641,32.633,-163.9561,16.1560,-6109.7750
C01347=-86.053,-13.053,32.146,-170.0298,32.5775,-6111.3748
C01348=-86.186,-8.933,31.951,-178.3732,35.7506,-6114.0825
C01349=-86.503,-4.570,31.943,179.8896,35.9073,-6116.9758
C01350=-86.627,0.000,31.948,180.0000,35.8947,-6120.0000
C01351=-86.503,4.570,31.943,-179.8896,35.9073,-6123.0242
C01352=-86.186,8.933,31.951,178.3732,35.7506,-6125.9175
C01353=-86.053,13.053,32.146,170.0298,32.5775,-6128.6252
C01354=-86.712,15.641,32.633,163.9561,16.1560,-6130.2250
C01355=-88.113,17.370,33.299,171.2911,4.6136,-6131.1519
C01356=-90.045,18.822,33.980,177.5928,0.9554,-6131.8065
C01357=-92.176,20.308,34.500,-179.3523,-0.3032,-6132.4248
C01358=-94.017,22.152,34.757,-179.2110,-0.7502,-6133.2580
C01359=-95.129,25.107,34.893,-179.6486,-0.7251,-6134.7847
C01360=-95.307,28.812,35.004,-179.8159,-0.8662,-6136.8204
C01361=-94.457,32.664,35.116,-179.9998,-0.0181,-6139.0758
C01362=-93.126,36.417,35.190,-179.9979,-0.0053,-6141.3580
C01363=-91.601,40.099,35.190,-179.9977,-0.0052,-6143.6417
C01364=-89.888,43.694,35.116,-179.9976,-0.0180,-6145.9241
C01365=-87.765,47.019,35.004,179.8142,-0.8665,-6148.1796
C01366=-85.019,49.513,34.893,179.6485,-0.7285,-6150.2155
C01367=-82.144,50.816,34.757,179.2111,-0.7508,-6151.7418
C01368=-79.538,50.818,34.500,179.3519,-0.3053,-6152.5751
C01369=-76.980,50.362,33.980,-177.5895,0.9541,-6153.1936
C01370=-74.588,50.022,33.299,-171.2890,4.6171,-6153.8475
C01371=-72.374,50.255,32.633,-163.9525,16.1553,-6154.7753
C01372=-70.079,51.619,32.146,-170.0305,32.5797,-6156.3747
C01373=-67.259,54.626,31.951,-178.3760,35.7490,-6159.0826
C01374=-64.399,57.935,31.943,179.8882,35.9085,-6161.9754
C01375=-61.254,61.254,31.948,180.0000,35.8962,-6165.0000
C01376=-57.936,64.398,31.943,-179.8875,35.9085,-6168.0237
C01377=-54.626,67.259,31.951,178.3760,35.7490,-6170.9174
C01378=-51.619,70.079,32.146,170.0305,32.5797,-6173.6253
C01379=-50.255,72.374,32.633,163.9525,16.1553,-6175.2247
C01380=-50.022,74.588,33.299,171.2890,4.6171,-6176.1525
C01381=-50.362,76.980,33.980,177.5895,0.9541,-6176.8064
C01382=-50.818,79.538,34.500,-179.3519,-0.3053,-6177.4249
C01383=-50.816,82.144,34.757,-179.2111,-0.7508,-6178.2582
C01384=-49.513,85.019,34.893,-179.6485,-0.7285,-6179.7845
C01385=-47.019,87.765,35.004,-179.8142,-0.8665,-6181.8204
C01386=-43.694,89.888,35.116,179.9976,-0.0180,-6184.0759
C01387=-40.099,91.601,35.190,179.9977,-0.0052,-6186.3583
C01388=-36.417,93.126,35.190,179.9979,-0.0053,-6188.6420
C01389=-32.664,94.457,35.116,179.9998,-0.0181,-6190.9242
C01390=-28.812,95.307,35.004,179.8159,-0.8662,-6193.1796
C01391=-25.107,95.129,34.893,179.6486,-0.7251,-6195.2153
C01392=-22.152,94.017,34.757,179.2110,-0.7502,-6196.7420
C01393=-20.308,92.176,34.500,179.3523,-0.3032,-6197.5752
C01394=-18.822,90.045,33.980,-177.5928,0.9554,-6198.1935
C01395=-17.370,88.113,33.299,-171.2911,4.6136,-6198.8481
C01396=-15.641,86.712,32.633,-163.9561,16.1560,-6199.7750
C01397=-13.053,86.053,32.146,-170.0298,32.5775,-6201.3748
C01398=-8.933,86.186,31.951,-178.3732,35.7506,-6204.0825
C01399=-4.570,86.503,31.943,179.8896,35.9073,-6206.9758
C01400=0.000,85.325,33.722,-180.0000,36.6281,-6210.0000
C01401=4.451,85.206,33.716,-179.8737,36.6409,-6212.9903
C01402=8.733,84.900,33.725,178.1463,36.4598,-6215.8729
C01403=12.808,84.808,33.943,168.8261,32.7893,-6218.5881
C01404=15.338,85.570,34.490,163.9088,14.2031,-6220.1621
C01405=17.019,87.137,35.239,172.4198,3.4506,-6221.0515
C01406=18.435,89.289,36.009,178.7364,0.4238,-6221.6656
C01407=19.887,91.675,36.600,-178.2531,-0.7002,-6222.2395
C01408=21.692,93.766,36.894,-178.4010,-1.3423,-6223.0258
C01409=24.671,95.076,37.049,-179.3934,-1.1510,-6224.5467
C01410=28.465,95.370,37.176,-179.7578,-1.0519,-6226.6187
C01411=32.445,94.529,37.304,-179.9997,-0.0362,-6228.9437
C01412=36.342,93.155,37.389,-179.9979,-0.0053,-6231.3119
C01413=40.172,91.569,37.389,-179.9977,-0.0052,-6233.6874
C01414=43.901,89.784,37.304,179.9971,-0.0333,-6236.0569
C01415=47.309,87.565,37.176,179.7616,-1.0536,-6238.3812
C01416=49.784,84.674,37.049,179.3922,-1.1484,-6240.4534
C01417=50.965,81.641,36.894,178.3995,-1.3439,-6241.9748
C01418=50.762,78.886,36.600,178.2560,-0.6999,-6242.7607
C01419=50.101,76.172,36.009,-178.7370,0.4261,-6243.3343
C01420=49.580,73.649,35.239,-172.4189,3.4541,-6243.9482
C01421=49.662,71.353,34.490,-163.9057,14.2058,-6244.8381
C01422=50.912,69.025,33.943,-168.8287,32.7883,-6246.4120
C01423=53.858,66.209,33.725,-178.1431,36.4603,-6249.1268
C01424=57.102,63.397,33.716,179.8751,36.6399,-6252.0095
C01425=60.334,60.334,33.722,-180.0000,36.6307,-6255.0000
C01426=63.397,57.102,33.716,-179.8751,36.6399,-6257.9905
C01427=66.209,53.858,33.725,178.1431,36.4603,-6260.8732
C01428=69.025,50.912,33.943,168.8287,32.7883,-6263.5880
C01429=71.353,49.662,34.490,163.9057,14.2058,-6265.1619
C01430=73.649,49.580,35.239,172.4189,3.4541,-6266.0518
C01431=76.172,50.101,36.009,178.7370,0.4261,-6266.6657
C01432=78.886,50.762,36.600,-178.2560,-0.6999,-6267.2393
C01433=81.641,50.965,36.894,-178.3995,-1.3439,-6268.0252
C01434=84.674,49.784,37.049,-179.3922,-1.1484,-6269.5466
C01435=87.565,47.309,37.176,-179.7616,-1.0536,-6271.6188
C01436=89.784,43.901,37.304,-179.9971,-0.0333,-6273.9431
C01437=91.569,40.172,37.389,179.9977,-0.0052,-6276.3126
C01438=93.155,36.342,37.389,179.9979,-0.0053,-6278.6881
C01439=94.529,32.445,37.304,179.9997,-0.0362,-6281.0563
C01440=95.370,28.465,37.176,179.7578,-1.0519,-6283.3813
C01441=95.076,24.671,37.049,179.3934,-1.1510,-6285.4533
C01442=93.766,21.692,36.894,178.4010,-1.3423,-6286.9742
C01443=91.675,19.887,36.600,178.2531,-0.7002,-6287.7605
C01444=89.289,18.435,36.009,-178.7364,0.4238,-6288.3344
C01445=87.137,17.019,35.239,-172.4198,3.4506,-6288.9485
C01446=85.570,15.338,34.490,-163.9088,14.2031,-6289.8379
C01447=84.808,12.808,33.943,-168.8261,32.7893,-6291.4119
C01448=84.900,8.733,33.725,-178.1463,36.4598,-6294.1271
C01449=85.206,4.451,33.716,179.8737,36.6409,-6297.0097
C01450=85.325,0.000,33.722,-180.0000,36.6281,-6300.0000
C01451=85.206,-4.451,33.716,-179.8737,36.6409,-6302.9903
C01452=84.900,-8.733,33.725,178.1463,36.4598,-6305.8729
C01453=84.808,-12.808,33.943,168.8327,32.7900,-6308.5881
C01454=85.570,-15.338,34.490,163.9088,14.2031,-6310.1621
C01455=87.137,-17.019,35.239,172.4198,3.4506,-6311.0515
C01456=89.289,-18.435,36.009,178.7364,0.4238,-6311.6656
C01457=91.675,-19.887,36.600,-178.2531,-0.7002,-6312.2395
C01458=93.766,-21.692,36.894,-178.4010,-1.3423,-6313.0258
C01459=95.076,-24.671,37.049,-179.3934,-1.1510,-6314.5467
C01460=95.370,-28.465,37.176,-179.7578,-1.0519,-6316.6187
C01461=94.529,-32.445,37.304,-179.9997,-0.0362,-6318.9437
C01462=93.155,-36.342,37.389,-179.9979,-0.0053,-6321.3119
C01463=91.569,-40.172,37.389,-179.9977,-0.0052,-6323.6874
C01464=89.784,-43.901,37.304,179.9971,-0.0333,-6326.0569
C01465=87.565,-47.309,37.176,179.7616,-1.0536,-6328.3812
C01466=84.674,-49.784,37.049,179.3922,-1.1484,-6330.4534
C01467=81.641,-50.965,36.894,178.3995,-1.3439,-6331.9748
C01468=78.886,-50.762,36.600,178.2560,-0.6999,-6332.7607
C01469=76.172,-50.101,36.009,-178.7370,0.4261,-6333.3343
C01470=73.649,-49.580,35.239,-172.4189,3.4541,-6333.9482
C01471=71.353,-49.662,34.490,-163.9057,14.2058,-6334.8381
C01472=69.025,-50.912,33.943,-168.8287,32.7883,-6336.4120
C01473=66.209,-53.858,33.725,-178.1431,36.4603,-6339.1268
C01474=63.397,-57.102,33.716,179.8751,36.6399,-6342.0095
C01475=60.334,-60.334,33.722,180.0000,36.6307,-6345.0000
C01476=57.102,-63.397,33.716,-179.8751,36.6399,-6347.9905
C01477=53.858,-66.209,33.725,178.1431,36.4603,-6350.8732
C01478=50.912,-69.025,33.943,168.8287,32.7883,-6353.5880
C01479=49.662,-71.353,34.490,163.9057,14.2058,-6355.1619
C01480=49.580,-73.649,35.239,172.4189,3.4541,-6356.0518
C01481=50.101,-76.172,36.009,178.7370,0.4261,-6356.6657
C01482=50.762,-78.886,36.600,-178.2560,-0.6999,-6357.2393
C01483=50.965,-81.641,36.894,-178.3995,-1.3439,-6358.0252
C01484=49.784,-84.674,37.049,-179.3922,-1.1484,-6359.5466
C01485=47.309,-87.565,37.176,-179.7616,-1.0536,-6361.6188
C01486=43.901,-89.784,37.304,-179.9971,-0.0333,-6363.9431
C01487=40.172,-91.569,37.389,179.9977,-0.0052,-6366.3126
C01488=36.342,-93.155,37.389,179.9979,-0.0053,-6368.6881
C01489=32.445,-94.529,37.304,179.9997,-0.0362,-6371.0563
C01490=28.465,-95.370,37.176,179.7578,-1.0519,-6373.3813
C01491=24.671,-95.076,37.049,179.3934,-1.1510,-6375.4533
C01492=21.692,-93.766,36.894,178.4010,-1.3423,-6376.9742
C01493=19.887,-91.675,36.600,178.2531,-0.7002,-6377.7605
C01494=18.435,-89.289,36.009,-178.7364,0.4238,-6378.3344
C01495=17.019,-87.137,35.239,-172.4198,3.4506,-6378.9485
C01496=15.338,-85.570,34.490,-163.9088,14.2031,-6379.8379
C01497=12.808,-84.808,33.943,-168.8261,32.7893,-6381.4119
C01498=8.733,-84.900,33.725,-178.1463,36.4598,-6384.1271
C01499=4.451,-85.206,33.716,179.8737,36.6409,-6387.0097
C01500=0.000,-85.325,33.722,180.0000,36.6281,-6390.0000
C01501=-4.451,-85.206,33.716,-179.8737,36.6409,-6392.9903
C01502=-8.733,-84.900,33.725,178.1463,36.4598,-6395.8729
C01503=-12.808,-84.808,33.943,168.8327,32.7900,-6398.5881
C01504=-15.338,-85.570,34.490,163.9088,14.2031,-6400.1621
C01505=-17.019,-87.137,35.239,172.4198,3.4506,-6401.0515
C01506=-18.435,-89.289,36.009,178.7364,0.4238,-6401.6656
C01507=-19.887,-91.675,36.600,-178.2531,-0.7002,-6402.2395
C01508=-21.692,-93.766,36.894,-178.4010,-1.3423,-6403.0258
C01509=-24.671,-95.076,37.049,-179.3934,-1.1510,-6404.5467
C01510=-28.465,-95.370,37.176,-179.7578,-1.0519,-6406.6187
C01511=-32.445,-94.529,37.304,-179.9997,-0.0362,-6408.9437
C01512=-36.342,-93.155,37.389,-179.9979,-0.0053,-6411.3119
C01513=-40.172,-91.569,37.389,-179.9977,-0.0052,-6413.6874
C01514=-43.901,-89.784,37.304,179.9971,-0.0333,-6416.0569
C01515=-47.309,-87.565,37.176,179.7616,-1.0536,-6418.3812
C01516=-49.784,-84.674,37.049,179.3922,-1.1484,-6420.4534
C01517=-50.965,-81.641,36.894,178.3995,-1.3439,-6421.9748
C01518=-50.762,-78.886,36.600,178.2560,-0.6999,-6422.7607
C01519=-50.101,-76.172,36.009,-178.7370,0.4261,-6423.3343
C01520=-49.580,-73.649,35.239,-172.4189,3.4541,-6423.9482
C01521=-49.662,-71.353,34.490,-163.9057,14.2058,-6424.8381
C01522=-50.912,-69.025,33.943,-168.8287,32.7883,-6426.4120
C01523=-53.858,-66.209,33.725,-178.1431,36.4603,-6429.1268
C01524=-57.102,-63.397,33.716,179.8751,36.6399,-6432.0095
C01525=-60.334,-60.334,33.722,-180.0000,36.6307,-6435.0000
C01526=-63.397,-57.102,33.716,-179.8751,36.6399,-6437.9905
C01527=-66.209,-53.858,33.725,178.1431,36.4603,-6440.8732
C01528=-69.025,-50.912,33.943,168.8287,32.7883,-6443.5880
C01529=-71.353,-49.662,34.490,163.9057,14.2058,-6445.1619
C01530=-73.649,-49.580,35.239,172.4189,3.4541,-6446.0518
C01531=-76.172,-50.101,36.009,178.7370,0.4261,-6446.6657
C01532=-78.886,-50.762,36.600,-178.2560,-0.6999,-6447.2393
C01533=-81.641,-50.965,36.894,-178.3995,-1.3439,-6448.0252
C01534=-84.674,-49.784,37.049,-179.3922,-1.1484,-6449.5466
C01535=-87.565,-47.309,37.176,-179.7616,-1.0536,-6451.6188
C01536=-89.784,-43.901,37.304,-179.9971,-0.0333,-6453.9431
C01537=-91.569,-40.172,37.389,179.9977,-0.0052,-6456.3126
C01538=-93.155,-36.342,37.389,179.9979,-0.0053,-6458.6881
C01539=-94.529,-32.445,37.304,179.9997,-0.0362,-6461.0563
C01540=-95.370,-28.465,37.176,179.7578,-1.0519,-6463.3813
C01541=-95.076,-24.671,37.049,179.3934,-1.1510,-6465.4533
C01542=-93.766,-21.692,36.894,178.4010,-1.3423,-6466.9742
C01543=-91.675,-19.887,36.600,178.2531,-0.7002,-6467.7605
C01544=-89.289,-18.435,36.009,-178.7364,0.4238,-6468.3344
C01545=-87.137,-17.019,35.239,-172.4198,3.4506,-6468.9485
C01546=-85.570,-15.338,34.490,-163.9088,14.2031,-6469.8379
C01547=-84.808,-12.808,33.943,-168.8261,32.7893,-6471.4119
C01548=-84.900,-8.733,33.725,-178.1463,36.4598,-6474.1271
C01549=-85.206,-4.451,33.716,179.8737,36.6409,-6477.0097
C01550=-85.325,0.000,33.722,-180.0000,36.6281,-6480.0000
C01551=-85.206,4.451,33.716,-179.8737,36.6409,-6482.9903
C01552=-84.900,8.733,33.725,178.1463,36.4598,-6485.8729
C01553=-84.808,12.808,33.943,168.8327,32.7900,-6488.5881
C01554=-85.570,15.338,34.490,163.9088,14.2031,-6490.1621
C01555=-87.137,17.019,35.239,172.4198,3.4506,-6491.0515
C01556=-89.289,18.435,36.009,178.7364,0.4238,-6491.6656
C01557=-91.675,19.887,36.600,-178.2531,-0.7002,-6492.2395
C01558=-93.766,21.692,36.894,-178.4010,-1.3423,-6493.0258
C01559=-95.076,24.671,37.049,-179.3934,-1.1510,-6494.5467
C01560=-95.370,28.465,37.176,-179.7578,-1.0519,-6496.6187
C01561=-94.529,32.445,37.304,-179.9997,-0.0362,-6498.9437
C01562=-93.155,36.342,37.389,-179.9979,-0.0053,-6501.3119
C01563=-91.569,40.172,37.389,-179.9977,-0.0052,-6503.6874
C01564=-89.784,43.901,37.304,179.9971,-0.0333,-6506.0569
C01565=-87.565,47.309,37.176,179.7616,-1.0536,-6508.3812
C01566=-84.674,49.784,37.049,179.3922,-1.1484,-6510.4534
C01567=-81.641,50.965,36.894,178.3995,-1.3439,-6511.9748
C01568=-78.886,50.762,36.600,178.2560,-0.6999,-6512.7607
C01569=-76.172,50.101,36.009,-178.7370,0.4261,-6513.3343
C01570=-73.649,49.580,35.239,-172.4189,3.4541,-6513.9482
C01571=-71.353,49.662,34.490,-163.9057,14.2058,-6514.8381
C01572=-69.025,50.912,33.943,-168.8287,32.7883,-6516.4120
C01573=-66.209,53.858,33.725,-178.1431,36.4603,-6519.1268
C01574=-63.397,57.102,33.716,179.8751,36.6399,-6522.0095
C01575=-60.334,60.334,33.722,-180.0000,36.6307,-6525.0000
C01576=-57.102,63.397,33.716,-179.8751,36.6399,-6527.9905
C01577=-53.858,66.209,33.725,178.1431,36.4603,-6530.8732
C01578=-50.912,69.025,33.943,168.8287,32.7883,-6533.5880
C01579=-49.662,71.353,34.490,163.9057,14.2058,-6535.1619
C01580=-49.580,73.649,35.239,172.4189,3.4541,-6536.0518
C01581=-50.101,76.172,36.009,178.7370,0.4261,-6536.6657
C01582=-50.762,78.886,36.600,-178.2560,-0.6999,-6537.2393
C01583=-50.965,81.641,36.894,-178.3995,-1.3439,-6538.0252
C01584=-49.784,84.674,37.049,-179.3922,-1.1484,-6539.5466
C01585=-47.309,87.565,37.176,-179.7616,-1.0536,-6541.6188
C01586=-43.901,89.784,37.304,-179.9971,-0.0333,-6543.9431
C01587=-40.172,91.569,37.389,179.9977,-0.0052,-6546.3126
C01588=-36.342,93.155,37.389,179.9979,-0.0053,-6548.6881
C01589=-32.445,94.529,37.304,179.9997,-0.0362,-6551.0563
C01590=-28.465,95.370,37.176,179.7578,-1.0519,-6553.3813
C01591=-24.671,95.076,37.049,179.3934,-1.1510,-6555.4533
C01592=-21.692,93.766,36.894,178.4010,-1.3423,-6556.9742
C01593=-19.887,91.675,36.600,178.2531,-0.7002,-6557.7605
C01594=-18.435,89.289,36.009,-178.7364,0.4238,-6558.3344
C01595=-17.019,87.137,35.239,-172.4198,3.4506,-6558.9485
C01596=-15.338,85.570,34.490,-163.9088,14.2031,-6559.8379
C01597=-12.808,84.808,33.943,-168.8327,32.7900,-6561.4119
C01598=-8.733,84.900,33.725,-178.1463,36.4598,-6564.1271
C01599=-4.451,85.206,33.716,179.8737,36.6409,-6567.0097
C01600=0.000,84.003,35.480,180.0000,37.2584,-6570.0000
C01601=4.330,83.888,35.473,-179.8571,37.2713,-6572.9548
C01602=8.530,83.594,35.484,177.9021,37.0692,-6575.8263
C01603=12.558,83.543,35.726,167.6478,32.8316,-6578.5486
C01604=15.030,84.409,36.333,164.2172,12.2420,-6580.0964
C01605=16.662,86.143,37.169,173.6165,2.5084,-6580.9471
C01606=18.041,88.518,38.031,179.8324,0.0477,-6581.5198
C01607=19.458,91.164,38.697,-177.2185,-0.9486,-6582.0484
C01608=21.221,93.510,39.027,-177.5538,-1.8150,-6582.7860
C01609=24.227,95.023,39.203,-179.1127,-1.5540,-6584.3034
C01610=28.112,95.435,39.346,-179.6955,-1.2364,-6586.4132
C01611=32.220,94.603,39.491,179.9985,-0.0489,-6588.8079
C01612=36.266,93.184,39.587,-179.9979,-0.0053,-6591.2653
C01613=40.247,91.535,39.587,179.9971,-0.0076,-6593.7346
C01614=44.111,89.678,39.491,179.9997,-0.0512,-6596.1917
C01615=47.604,87.360,39.346,179.6949,-1.2364,-6598.5867
C01616=50.060,84.322,39.203,179.1149,-1.5518,-6600.6966
C01617=51.116,81.128,39.027,177.5559,-1.8116,-6602.2136
C01618=50.704,78.221,38.697,177.2195,-0.9491,-6602.9519
C01619=49.835,75.348,38.031,-179.8330,0.0487,-6603.4806
C01620=49.130,72.694,37.169,-173.6149,2.5069,-6604.0527
C01621=49.058,70.314,36.333,-164.2153,12.2381,-6604.9034
C01622=50.194,67.954,35.726,-167.6473,32.8330,-6606.4513
C01623=53.078,65.141,35.484,-177.8974,37.0682,-6609.1737
C01624=56.256,62.380,35.473,179.8597,37.2688,-6612.0450
C01625=59.399,59.399,35.480,180.0000,37.2595,-6615.0000
C01626=62.380,56.256,35.473,-179.8597,37.2688,-6617.9550
C01627=65.141,53.078,35.484,177.8974,37.0682,-6620.8263
C01628=67.954,50.194,35.726,167.6473,32.8330,-6623.5487
C01629=70.314,49.058,36.333,164.2153,12.2381,-6625.0966
C01630=72.694,49.130,37.169,173.6149,2.5069,-6625.9473
C01631=75.348,49.835,38.031,179.8330,0.0487,-6626.5194
C01632=78.221,50.704,38.697,-177.2195,-0.9491,-6627.0481
C01633=81.128,51.116,39.027,-177.5559,-1.8116,-6627.7864
C01634=84.322,50.060,39.203,-179.1149,-1.5518,-6629.3034
C01635=87.360,47.604,39.346,-179.6949,-1.2364,-6631.4133
C01636=89.678,44.111,39.491,-179.9997,-0.0512,-6633.8083
C01637=91.535,40.247,39.587,-179.9971,-0.0076,-6636.2654
C01638=93.184,36.266,39.587,179.9979,-0.0053,-6638.7347
C01639=94.603,32.220,39.491,-179.9985,-0.0489,-6641.1921
C01640=95.435,28.112,39.346,179.6955,-1.2364,-6643.5868
C01641=95.023,24.227,39.203,179.1127,-1.5540,-6645.6966
C01642=93.510,21.221,39.027,177.5538,-1.8150,-6647.2140
C01643=91.164,19.458,38.697,177.2185,-0.9486,-6647.9516
C01644=88.518,18.041,38.031,-179.8324,0.0477,-6648.4802
C01645=86.143,16.662,37.169,-173.6165,2.5084,-6649.0529
C01646=84.409,15.030,36.333,-164.2172,12.2420,-6649.9036
C01647=83.543,12.558,35.726,-167.6478,32.8316,-6651.4514
C01648=83.594,8.530,35.484,-177.9021,37.0692,-6654.1737
C01649=83.888,4.330,35.473,179.8571,37.2713,-6657.0452
C01650=84.003,0.000,35.480,-180.0000,37.2584,-6660.0000
C01651=83.888,-4.330,35.473,-179.8571,37.2713,-6662.9548
C01652=83.594,-8.530,35.484,177.8949,37.0687,-6665.8263
C01653=83.543,-12.558,35.726,167.6478,32.8316,-6668.5486
C01654=84.409,-15.030,36.333,164.2172,12.2420,-6670.0964
C01655=86.143,-16.662,37.169,173.6165,2.5084,-6670.9471
C01656=88.518,-18.041,38.031,179.8324,0.0477,-6671.5198
C01657=91.164,-19.458,38.697,-177.2185,-0.9486,-6672.0484
C01658=93.510,-21.221,39.027,-177.5538,-1.8150,-6672.7860
C01659=95.023,-24.227,39.203,-179.1127,-1.5540,-6674.3034
C01660=95.435,-28.112,39.346,-179.6955,-1.2364,-6676.4132
C01661=94.603,-32.220,39.491,179.9985,-0.0489,-6678.8079
C01662=93.184,-36.266,39.587,-179.9979,-0.0053,-6681.2653
C01663=91.535,-40.247,39.587,179.9971,-0.0076,-6683.7346
C01664=89.678,-44.111,39.491,179.9997,-0.0512,-6686.1917
C01665=87.360,-47.604,39.346,179.6949,-1.2364,-6688.5867
C01666=84.322,-50.060,39.203,179.1149,-1.5518,-6690.6966
C01667=81.128,-51.116,39.027,177.5559,-1.8116,-6692.2136
C01668=78.221,-50.704,38.697,177.2195,-0.9491,-6692.9519
C01669=75.348,-49.835,38.031,-179.8330,0.0487,-6693.4806
C01670=72.694,-49.130,37.169,-173.6149,2.5069,-6694.0527
C01671=70.314,-49.058,36.333,-164.2153,12.2381,-6694.9034
C01672=67.954,-50.194,35.726,-167.6473,32.8330,-6696.4513
C01673=65.141,-53.078,35.484,-177.8974,37.0682,-6699.1737
C01674=62.380,-56.256,35.473,179.8597,37.2688,-6702.0450
C01675=59.399,-59.399,35.480,-180.0000,37.2595,-6705.0000
C01676=56.256,-62.380,35.473,-179.8597,37.2688,-6707.9550
C01677=53.078,-65.141,35.484,177.8974,37.0682,-6710.8263
C01678=50.194,-67.954,35.726,167.6473,32.8330,-6713.5487
C01679=49.058,-70.314,36.333,164.2153,12.2381,-6715.0966
C01680=49.130,-72.694,37.169,173.6149,2.5069,-6715.9473
C01681=49.835,-75.348,38.031,179.8330,0.0487,-6716.5194
C01682=50.704,-78.221,38.697,-177.2195,-0.9491,-6717.0481
C01683=51.116,-81.128,39.027,-177.5559,-1.8116,-6717.7864
C01684=50.060,-84.322,39.203,-179.1149,-1.5518,-6719.3034
C01685=47.604,-87.360,39.346,-179.6949,-1.2364,-6721.4133
C01686=44.111,-89.678,39.491,-179.9997,-0.0512,-6723.8083
C01687=40.247,-91.535,39.587,-179.9971,-0.0076,-6726.2654
C01688=36.266,-93.184,39.587,179.9979,-0.0053,-6728.7347
C01689=32.220,-94.603,39.491,-179.9985,-0.0489,-6731.1921
C01690=28.112,-95.435,39.346,179.6955,-1.2364,-6733.5868
C01691=24.227,-95.023,39.203,179.1127,-1.5540,-6735.6966
C01692=21.221,-93.510,39.027,177.5538,-1.8150,-6737.2140
C01693=19.458,-91.164,38.697,177.2185,-0.9486,-6737.9516
C01694=18.041,-88.518,38.031,-179.8324,0.0477,-6738.4802
C01695=16.662,-86.143,37.169,-173.6165,2.5084,-6739.0529
C01696=15.030,-84.409,36.333,-164.2172,12.2420,-6739.9036
C01697=12.558,-83.543,35.726,-167.6478,32.8316,-6741.4514
C01698=8.530,-83.594,35.484,-177.9021,37.0692,-6744.1737
C01699=4.330,-83.888,35.473,179.8571,37.2713,-6747.0452
C01700=0.000,-84.003,35.480,-180.0000,37.2584,-6750.0000
C01701=-4.330,-83.888,35.473,-179.8571,37.2713,-6752.9548
C01702=-8.530,-83.594,35.484,177.8949,37.0687,-6755.8263
C01703=-12.558,-83.543,35.726,167.6478,32.8316,-6758.5486
C01704=-15.030,-84.409,36.333,164.2172,12.2420,-6760.0964
C01705=-16.662,-86.143,37.169,173.6165,2.5084,-6760.9471
C01706=-18.041,-88.518,38.031,179.8324,0.0477,-6761.5198
C01707=-19.458,-91.164,38.697,-177.2185,-0.9486,-6762.0484
C01708=-21.221,-93.510,39.027,-177.5538,-1.8150,-6762.7860
C01709=-24.227,-95.023,39.203,-179.1127,-1.5540,-6764.3034
C01710=-28.112,-95.435,39.346,-179.6955,-1.2364,-6766.4132
C01711=-32.220,-94.603,39.491,179.9985,-0.0489,-6768.8079
C01712=-36.266,-93.184,39.587,-179.9979,-0.0053,-6771.2653
C01713=-40.247,-91.535,39.587,179.9971,-0.0076,-6773.7346
C01714=-44.111,-89.678,39.491,179.9997,-0.0512,-6776.1917
C01715=-47.604,-87.360,39.346,179.6949,-1.2364,-6778.5867
C01716=-50.060,-84.322,39.203,179.1149,-1.5518,-6780.6966
C01717=-51.116,-81.128,39.027,177.5559,-1.8116,-6782.2136
C01718=-50.704,-78.221,38.697,177.2195,-0.9491,-6782.9519
C01719=-49.835,-75.348,38.031,-179.8330,0.0487,-6783.4806
C01720=-49.130,-72.694,37.169,-173.6149,2.5069,-6784.0527
C01721=-49.058,-70.314,36.333,-164.2153,12.2381,-6784.9034
C01722=-50.194,-67.954,35.726,-167.6473,32.8330,-6786.4513
C01723=-53.078,-65.141,35.484,-177.8974,37.0682,-6789.1737
C01724=-56.256,-62.380,35.473,179.8597,37.2688,-6792.0450
C01725=-59.399,-59.399,35.480,-180.0000,37.2595,-6795.0000
C01726=-62.380,-56.256,35.473,-179.8597,37.2688,-6797.9550
C01727=-65.141,-53.078,35.484,177.8974,37.0682,-6800.8263
C01728=-67.954,-50.194,35.726,167.6473,32.8330,-6803.5487
C01729=-70.314,-49.058,36.333,164.2153,12.2381,-6805.0966
C01730=-72.694,-49.130,37.169,173.6149,2.5069,-6805.9473
C01731=-75.348,-49.835,38.031,179.8330,0.0487,-6806.5194
C01732=-78.221,-50.704,38.697,-177.2195,-0.9491,-6807.0481
C01733=-81.128,-51.116,39.027,-177.5559,-1.8116,-6807.7864
C01734=-84.322,-50.060,39.203,-179.1149,-1.5518,-6809.3034
C01735=-87.360,-47.604,39.346,-179.6949,-1.2364,-6811.4133
C01736=-89.678,-44.111,39.491,-179.9997,-0.0512,-6813.8083
C01737=-91.535,-40.247,39.587,-179.9971,-0.0076,-6816.2654
C01738=-93.184,-36.266,39.587,179.9979,-0.0053,-6818.7347
C01739=-94.603,-32.220,39.491,-179.9985,-0.0489,-6821.1921
C01740=-95.435,-28.112,39.346,179.6955,-1.2364,-6823.5868
C01741=-95.023,-24.227,39.203,179.1127,-1.5540,-6825.6966
C01742=-93.510,-21.221,39.027,177.5538,-1.8150,-6827.2140
C01743=-91.164,-19.458,38.697,177.2185,-0.9486,-6827.9516
C01744=-88.518,-18.041,38.031,-179.8324,0.0477,-6828.4802
C01745=-86.143,-16.662,37.169,-173.6165,2.5084,-6829.0529
